LIN {X 0,Y 542.795,Z 373.704,A -85,B 0,C 180,E1 23564.562,E2 23564.562} C_VEL
LIN {X 0,Y 545.816,Z 376.25,A -85,B 0,C 180,E1 23563.586,E2 23563.586} C_VEL
LIN {X 0,Y 548.815,Z 380.332,A -85,B 0,C 180,E1 23562.615,E2 23562.615} C_VEL
LIN {X 0,Y 551.245,Z 382.532,A -85,B 0,C 180,E1 23561.903,E2 23561.903} C_VEL
LIN {X 0,Y 554.687,Z 386.919,A -85,B 0,C 180,E1 23560.902,E2 23560.902} C_VEL
LIN {X 0,Y 556.558,Z 388.828,A -85,B 0,C 180,E1 23560.396,E2 23560.396} C_VEL
LIN {X 0,Y 560.439,Z 393.498,A -85,B 0,C 180,E1 23559.368,E2 23559.368} C_VEL
LIN {X 0,Y 566.505,Z 400.97,A -85,B 0,C 180,E1 23557.862,E2 23557.862} C_VEL
LIN {X 0,Y 571.785,Z 407.602,A -85,B 0,C 180,E1 23556.639,E2 23556.639} C_VEL
LIN {X 0,Y 577.51,Z 414.886,A -85,B 0,C 180,E1 23555.392,E2 23555.392} C_VEL
LIN {X 0,Y 587.049,Z 428.51,A -85,B 0,C 180,E1 23553.442,E2 23553.442} C_VEL
LIN {X 0,Y 595.115,Z 441.003,A -85,B 0,C 180,E1 23551.909,E2 23551.909} C_VEL
LIN {X 0,Y 595.96,Z 442.638,A -85,B 0,C 180,E1 23551.748,E2 23551.748} C_VEL
LIN {X 0,Y 586.943,Z 655.568,A -85,B 0,C 180,E1 23548.557,E2 23548.557} C_VEL
LIN {X 0,Y 580.387,Z 818.11,A -85,B 0,C 180,E1 23546.144,E2 23546.144} C_VEL
LIN {X 0,Y 578.548,Z 843.182,A -85,B 0,C 180,E1 23545.671,E2 23545.671} C_VEL
LIN {X 0,Y 575.71,Z 870.919,A -85,B 0,C 180,E1 23544.956,E2 23544.956} C_VEL
LIN {X 0,Y 573.073,Z 892.207,A -85,B 0,C 180,E1 23544.266,E2 23544.266} C_VEL
LIN {X 0,Y 570.199,Z 912.697,A -85,B 0,C 180,E1 23543.475,E2 23543.475} C_VEL
LIN {X 0,Y 567.095,Z 932.487,A -85,B 0,C 180,E1 23542.588,E2 23542.588} C_VEL
LIN {X 0,Y 564.019,Z 950.451,A -85,B 0,C 180,E1 23541.669,E2 23541.669} C_VEL
LIN {X 0,Y 562.069,Z 957.506,A -85,B 0,C 180,E1 23541.362,E2 23541.362} C_VEL
LIN {X 0,Y 554.369,Z 974.984,A -85,B 0,C 180,E1 23540.75,E2 23540.75} C_VEL
LIN {X 0,Y 552.285,Z 981.526,A -85,B 0,C 180,E1 23540.385,E2 23540.385} C_VEL
LIN {X 0,Y 548.266,Z 1000.587,A -85,B 0,C 180,E1 23539.025,E2 23539.025} C_VEL
LIN {X 0,Y 544.207,Z 1019.207,A -85,B 0,C 180,E1 23537.533,E2 23537.533} C_VEL
LIN {X 0,Y 539.48,Z 1040.477,A -85,B 0,C 180,E1 23535.6,E2 23535.6} C_VEL
LIN {X 0,Y 534.654,Z 1061.325,A -85,B 0,C 180,E1 23533.414,E2 23533.414} C_VEL
LIN {X 0,Y 530.182,Z 1080.685,A -85,B 0,C 180,E1 23531.091,E2 23531.091} C_VEL
LIN {X 0,Y 526.071,Z 1099.032,A -85,B 0,C 180,E1 23528.565,E2 23528.565} C_VEL
LIN {X 0,Y 522.347,Z 1116.161,A -85,B 0,C 180,E1 23525.855,E2 23525.855} C_VEL
LIN {X 0,Y 519.741,Z 1129.22,A -85,B 0,C 180,E1 23523.512,E2 23523.512} C_VEL
LIN {X 0,Y 517.517,Z 1141.407,A -85,B 0,C 180,E1 23521.054,E2 23521.054} C_VEL
LIN {X 0,Y 515.395,Z 1154.516,A -85,B 0,C 180,E1 23518,E2 23518} C_VEL
LIN {X 0,Y 514.05,Z 1164.255,A -85,B 0,C 180,E1 23515.335,E2 23515.335} C_VEL
LIN {X 0,Y 513.094,Z 1172.905,A -85,B 0,C 180,E1 23512.575,E2 23512.575} C_VEL
LIN {X 0,Y 512.416,Z 1180.779,A -85,B 0,C 180,E1 23509.491,E2 23509.491} C_VEL
LIN {X 0,Y 512.131,Z 1185.993,A -85,B 0,C 180,E1 23506.912,E2 23506.912} C_VEL
LIN {X 0,Y 511.987,Z 1189.961,A -85,B 0,C 180,E1 23504.379,E2 23504.379} C_VEL
LIN {X 0,Y 511.919,Z 1193.03,A -85,B 0,C 180,E1 23501.606,E2 23501.606} C_VEL
LIN {X 0,Y 511.91,Z 1194.672,A -85,B 0,C 180,E1 23498.65,E2 23498.65} C_VEL
LIN {X 0,Y 511.913,Z 1194.851,A -85,B 0,C 180,E1 23496.167,E2 23496.167} C_VEL
LIN {X 0,Y 511.909,Z 1193.96,A -85,B 0,C 180,E1 23493.696,E2 23493.696} C_VEL
LIN {X 0,Y 511.935,Z 1191.975,A -85,B 0,C 180,E1 23491.231,E2 23491.231} C_VEL
LIN {X 0,Y 512.028,Z 1188.452,A -85,B 0,C 180,E1 23488.433,E2 23488.433} C_VEL
LIN {X 0,Y 512.288,Z 1182.928,A -85,B 0,C 180,E1 23485.41,E2 23485.41} C_VEL
LIN {X 0,Y 512.716,Z 1176.911,A -85,B 0,C 180,E1 23482.83,E2 23482.83} C_VEL
LIN {X 0,Y 513.428,Z 1169.662,A -85,B 0,C 180,E1 23480.246,E2 23480.246} C_VEL
LIN {X 0,Y 514.741,Z 1159.044,A -85,B 0,C 180,E1 23477.092,E2 23477.092} C_VEL
LIN {X 0,Y 516.276,Z 1148.691,A -85,B 0,C 180,E1 23474.499,E2 23474.499} C_VEL
LIN {X 0,Y 518.205,Z 1137.424,A -85,B 0,C 180,E1 23472.018,E2 23472.018} C_VEL
LIN {X 0,Y 521.153,Z 1122.163,A -85,B 0,C 180,E1 23469.093,E2 23469.093} C_VEL
LIN {X 0,Y 524.187,Z 1107.393,A -85,B 0,C 180,E1 23466.625,E2 23466.625} C_VEL
LIN {X 0,Y 527.705,Z 1091.651,A -85,B 0,C 180,E1 23464.285,E2 23464.285} C_VEL
LIN {X 0,Y 532.183,Z 1072.006,A -85,B 0,C 180,E1 23461.741,E2 23461.741} C_VEL
LIN {X 0,Y 536.871,Z 1051.612,A -85,B 0,C 180,E1 23459.441,E2 23459.441} C_VEL
LIN {X 0,Y 541.664,Z 1030.618,A -85,B 0,C 180,E1 23457.384,E2 23457.384} C_VEL
LIN {X 0,Y 546.846,Z 1007.416,A -85,B 0,C 180,E1 23455.409,E2 23455.409} C_VEL
LIN {X 0,Y 551.213,Z 986.563,A -85,B 0,C 180,E1 23453.877,E2 23453.877} C_VEL
LIN {X 0,Y 554.892,Z 968.037,A -85,B 0,C 180,E1 23452.675,E2 23452.675} C_VEL
LIN {X 0,Y 558.395,Z 949.059,A -85,B 0,C 180,E1 23451.586,E2 23451.586} C_VEL
LIN {X 0,Y 561.883,Z 928.574,A -85,B 0,C 180,E1 23450.56,E2 23450.56} C_VEL
LIN {X 0,Y 565.837,Z 903.019,A -85,B 0,C 180,E1 23449.471,E2 23449.471} C_VEL
LIN {X 0,Y 569.101,Z 877.277,A -85,B 0,C 180,E1 23448.59,E2 23448.59} C_VEL
LIN {X 0,Y 571.431,Z 855.733,A -85,B 0,C 180,E1 23447.989,E2 23447.989} C_VEL
LIN {X 0,Y 573.333,Z 834.31,A -85,B 0,C 180,E1 23447.511,E2 23447.511} C_VEL
LIN {X 0,Y 574.879,Z 810.042,A -85,B 0,C 180,E1 23447.093,E2 23447.093} C_VEL
LIN {X 0,Y 582.975,Z 592.298,A -85,B 0,C 180,E1 23443.915,E2 23443.915} C_VEL
LIN {X 0,Y 588.599,Z 446.247,A -85,B 0,C 180,E1 23441.753,E2 23441.753} C_VEL
LIN {X 0,Y 572.418,Z 422.974,A -85,B 0,C 180,E1 23439.029,E2 23439.029} C_VEL
LIN {X 0,Y 564.92,Z 412.761,A -85,B 0,C 180,E1 23437.668,E2 23437.668} C_VEL
LIN {X 0,Y 556.568,Z 402.056,A -85,B 0,C 180,E1 23436.067,E2 23436.067} C_VEL
LIN {X 0,Y 548.839,Z 392.277,A -85,B 0,C 180,E1 23434.481,E2 23434.481} C_VEL
LIN {X 0,Y 543.88,Z 386.332,A -85,B 0,C 180,E1 23433.409,E2 23433.409} C_VEL
LIN {X 0,Y 539.41,Z 380.867,A -85,B 0,C 180,E1 23432.392,E2 23432.392} C_VEL
LIN {X 0,Y 535.79,Z 376.492,A -85,B 0,C 180,E1 23431.534,E2 23431.534} C_VEL
LIN {X 0,Y 534.25,Z 374.853,A -85,B 0,C 180,E1 23431.164,E2 23431.164} C_VEL
LIN {X 0,Y 530.972,Z 370.926,A -85,B 0,C 180,E1 23430.342,E2 23430.342} C_VEL
LIN {X 0,Y 529.918,Z 369.476,A -85,B 0,C 180,E1 23430.064,E2 23430.064} C_VEL
LIN {X 0,Y 526.592,Z 366.343,A -85,B 0,C 180,E1 23429.209,E2 23429.209} C_VEL
LIN {X 0,Y 524.818,Z 363.288,A -85,B 0,C 180,E1 23428.693,E2 23428.693} C_VEL
LIN {X 0,Y 521.507,Z 360.788,A -85,B 0,C 180,E1 23427.8,E2 23427.8} C_VEL
LIN {X 0,Y 519.538,Z 357.406,A -85,B 0,C 180,E1 23427.184,E2 23427.184} C_VEL
LIN {X 0,Y 519.072,Z 356.737,A -85,B 0,C 180,E1 23427.04,E2 23427.04} C_VEL
LIN {X 0,Y 515.845,Z 354.704,A -85,B 0,C 180,E1 23426.104,E2 23426.104} C_VEL
LIN {X 0,Y 514.186,Z 351.972,A -85,B 0,C 180,E1 23425.542,E2 23425.542} C_VEL
LIN {X 0,Y 513.777,Z 350.215,A -85,B 0,C 180,E1 23425.351,E2 23425.351} C_VEL
LIN {X 0,Y 513.713,Z 350.161,A -85,B 0,C 180,E1 23422.065,E2 23422.065} C_VEL
LIN {X 0,Y 513.745,Z 350.236,A -85,B 0,C 180,E1 23418.614,E2 23418.614} C_VEL
LIN {X 0,Y 513.754,Z 350.233,A -85,B 0,C 180,E1 23415.349,E2 23415.349} C_VEL
LIN {X 0,Y 513.723,Z 350.235,A -85,B 0,C 180,E1 23412.021,E2 23412.021} C_VEL
LIN {X 0,Y 513.776,Z 350.224,A -85,B 0,C 180,E1 23408.619,E2 23408.619} C_VEL
LIN {X 0,Y 513.734,Z 350.224,A -85,B 0,C 180,E1 23405.361,E2 23405.361} C_VEL
LIN {X 0,Y 513.728,Z 350.224,A -85,B 0,C 180,E1 23401.896,E2 23401.896} C_VEL
LIN {X 0,Y 513.784,Z 350.213,A -85,B 0,C 180,E1 23398.662,E2 23398.662} C_VEL
LIN {X 0,Y 513.727,Z 350.218,A -85,B 0,C 180,E1 23395.311,E2 23395.311} C_VEL
LIN {X 0,Y 513.743,Z 350.219,A -85,B 0,C 180,E1 23391.832,E2 23391.832} C_VEL
LIN {X 0,Y 513.764,Z 350.175,A -85,B 0,C 180,E1 23388.55,E2 23388.55} C_VEL
LIN {X 0,Y 513.725,Z 350.191,A -85,B 0,C 180,E1 23385.228,E2 23385.228} C_VEL
LIN {X 0,Y 513.781,Z 350.168,A -85,B 0,C 180,E1 23381.975,E2 23381.975} C_VEL
LIN {X 0,Y 513.776,Z 350.304,A -85,B 0,C 180,E1 23381.74,E2 23381.74} C_VEL
LIN {X 0,Y 514.652,Z 353.02,A -85,B 0,C 180,E1 23381.391,E2 23381.391} C_VEL
LIN {X 0,Y 516.89,Z 355.586,A -85,B 0,C 180,E1 23380.683,E2 23380.683} C_VEL
LIN {X 0,Y 519.415,Z 357.122,A -85,B 0,C 180,E1 23379.961,E2 23379.961} C_VEL
LIN {X 0,Y 521.3,Z 360.559,A -85,B 0,C 180,E1 23379.363,E2 23379.363} C_VEL
LIN {X 0,Y 524.371,Z 363.099,A -85,B 0,C 180,E1 23378.524,E2 23378.524} C_VEL
LIN {X 0,Y 525.111,Z 363.904,A -85,B 0,C 180,E1 23378.321,E2 23378.321} C_VEL
LIN {X 0,Y 527.649,Z 367.603,A -85,B 0,C 180,E1 23377.611,E2 23377.611} C_VEL
LIN {X 0,Y 530.517,Z 370.117,A -85,B 0,C 180,E1 23376.887,E2 23376.887} C_VEL
LIN {X 0,Y 533.502,Z 374.128,A -85,B 0,C 180,E1 23376.12,E2 23376.12} C_VEL
LIN {X 0,Y 535.754,Z 376.327,A -85,B 0,C 180,E1 23375.582,E2 23375.582} C_VEL
LIN {X 0,Y 545.223,Z 388.341,A -85,B 0,C 180,E1 23373.389,E2 23373.389} C_VEL
LIN {X 0,Y 553.809,Z 399.693,A -85,B 0,C 180,E1 23371.563,E2 23371.563} C_VEL
LIN {X 0,Y 562.926,Z 412.152,A -85,B 0,C 180,E1 23369.764,E2 23369.764} C_VEL
LIN {X 0,Y 575.646,Z 430.28,A -85,B 0,C 180,E1 23367.45,E2 23367.45} C_VEL
LIN {X 0,Y 588.662,Z 449.546,A -85,B 0,C 180,E1 23365.278,E2 23365.278} C_VEL
LIN {X 0,Y 580.389,Z 665.721,A -85,B 0,C 180,E1 23362.096,E2 23362.096} C_VEL
LIN {X 0,Y 574.374,Z 825.899,A -85,B 0,C 180,E1 23359.751,E2 23359.751} C_VEL
LIN {X 0,Y 572.583,Z 850.667,A -85,B 0,C 180,E1 23359.295,E2 23359.295} C_VEL
LIN {X 0,Y 569.722,Z 879.093,A -85,B 0,C 180,E1 23358.578,E2 23358.578} C_VEL
LIN {X 0,Y 567.068,Z 900.639,A -85,B 0,C 180,E1 23357.891,E2 23357.891} C_VEL
LIN {X 0,Y 564.208,Z 921.045,A -85,B 0,C 180,E1 23357.115,E2 23357.115} C_VEL
LIN {X 0,Y 560.986,Z 941.539,A -85,B 0,C 180,E1 23356.206,E2 23356.206} C_VEL
LIN {X 0,Y 556.988,Z 964.689,A -85,B 0,C 180,E1 23355.013,E2 23355.013} C_VEL
LIN {X 0,Y 552.164,Z 989.777,A -85,B 0,C 180,E1 23353.48,E2 23353.48} C_VEL
LIN {X 0,Y 548.264,Z 1008.64,A -85,B 0,C 180,E1 23352.153,E2 23352.153} C_VEL
LIN {X 0,Y 544.316,Z 1026.981,A -85,B 0,C 180,E1 23350.7,E2 23350.7} C_VEL
LIN {X 0,Y 540.243,Z 1045.39,A -85,B 0,C 180,E1 23349.063,E2 23349.063} C_VEL
LIN {X 0,Y 535.325,Z 1067.373,A -85,B 0,C 180,E1 23346.838,E2 23346.838} C_VEL
LIN {X 0,Y 531.26,Z 1085.19,A -85,B 0,C 180,E1 23344.768,E2 23344.768} C_VEL
LIN {X 0,Y 528.053,Z 1099.503,A -85,B 0,C 180,E1 23342.917,E2 23342.917} C_VEL
LIN {X 0,Y 525.031,Z 1113.29,A -85,B 0,C 180,E1 23340.943,E2 23340.943} C_VEL
LIN {X 0,Y 522.121,Z 1127.167,A -85,B 0,C 180,E1 23338.729,E2 23338.729} C_VEL
LIN {X 0,Y 519.005,Z 1143.116,A -85,B 0,C 180,E1 23335.81,E2 23335.81} C_VEL
LIN {X 0,Y 516.929,Z 1154.738,A -85,B 0,C 180,E1 23333.36,E2 23333.36} C_VEL
LIN {X 0,Y 515.373,Z 1164.516,A -85,B 0,C 180,E1 23331.033,E2 23331.033} C_VEL
LIN {X 0,Y 514.198,Z 1173.103,A -85,B 0,C 180,E1 23328.714,E2 23328.714} C_VEL
LIN {X 0,Y 513.172,Z 1181.977,A -85,B 0,C 180,E1 23325.945,E2 23325.945} C_VEL
LIN {X 0,Y 512.473,Z 1190.05,A -85,B 0,C 180,E1 23322.851,E2 23322.851} C_VEL
LIN {X 0,Y 512.147,Z 1195.486,A -85,B 0,C 180,E1 23320.233,E2 23320.233} C_VEL
LIN {X 0,Y 511.999,Z 1199.358,A -85,B 0,C 180,E1 23317.857,E2 23317.857} C_VEL
LIN {X 0,Y 511.932,Z 1202.314,A -85,B 0,C 180,E1 23315.379,E2 23315.379} C_VEL
LIN {X 0,Y 511.912,Z 1204.305,A -85,B 0,C 180,E1 23312.687,E2 23312.687} C_VEL
LIN {X 0,Y 511.897,Z 1204.939,A -85,B 0,C 180,E1 23309.664,E2 23309.664} C_VEL
LIN {X 0,Y 511.916,Z 1204.1,A -85,B 0,C 180,E1 23306.977,E2 23306.977} C_VEL
LIN {X 0,Y 511.933,Z 1202.199,A -85,B 0,C 180,E1 23304.508,E2 23304.508} C_VEL
LIN {X 0,Y 512.006,Z 1199.197,A -85,B 0,C 180,E1 23302.03,E2 23302.03} C_VEL
LIN {X 0,Y 512.169,Z 1195.073,A -85,B 0,C 180,E1 23299.54,E2 23299.54} C_VEL
LIN {X 0,Y 512.613,Z 1188.472,A -85,B 0,C 180,E1 23296.464,E2 23296.464} C_VEL
LIN {X 0,Y 513.312,Z 1180.562,A -85,B 0,C 180,E1 23293.594,E2 23293.594} C_VEL
LIN {X 0,Y 514.249,Z 1172.698,A -85,B 0,C 180,E1 23291.17,E2 23291.17} C_VEL
LIN {X 0,Y 515.439,Z 1164.061,A -85,B 0,C 180,E1 23288.85,E2 23288.85} C_VEL
LIN {X 0,Y 517.113,Z 1153.715,A -85,B 0,C 180,E1 23286.407,E2 23286.407} C_VEL
LIN {X 0,Y 519.812,Z 1138.894,A -85,B 0,C 180,E1 23283.373,E2 23283.373} C_VEL
LIN {X 0,Y 522.451,Z 1125.546,A -85,B 0,C 180,E1 23281.001,E2 23281.001} C_VEL
LIN {X 0,Y 525.203,Z 1112.507,A -85,B 0,C 180,E1 23278.941,E2 23278.941} C_VEL
LIN {X 0,Y 528.242,Z 1098.637,A -85,B 0,C 180,E1 23276.967,E2 23276.967} C_VEL
LIN {X 0,Y 532.231,Z 1080.973,A -85,B 0,C 180,E1 23274.713,E2 23274.713} C_VEL
LIN {X 0,Y 536.861,Z 1060.276,A -85,B 0,C 180,E1 23272.415,E2 23272.415} C_VEL
LIN {X 0,Y 540.77,Z 1042.882,A -85,B 0,C 180,E1 23270.709,E2 23270.709} C_VEL
LIN {X 0,Y 544.733,Z 1024.943,A -85,B 0,C 180,E1 23269.135,E2 23269.135} C_VEL
LIN {X 0,Y 549.73,Z 1001.929,A -85,B 0,C 180,E1 23267.351,E2 23267.351} C_VEL
LIN {X 0,Y 554.397,Z 978.674,A -85,B 0,C 180,E1 23265.809,E2 23265.809} C_VEL
LIN {X 0,Y 558.111,Z 959.029,A -85,B 0,C 180,E1 23264.665,E2 23264.665} C_VEL
LIN {X 0,Y 561.651,Z 938.954,A -85,B 0,C 180,E1 23263.643,E2 23263.643} C_VEL
LIN {X 0,Y 565.072,Z 917.752,A -85,B 0,C 180,E1 23262.71,E2 23262.71} C_VEL
LIN {X 0,Y 568.897,Z 890.935,A -85,B 0,C 180,E1 23261.725,E2 23261.725} C_VEL
LIN {X 0,Y 571.809,Z 865.86,A -85,B 0,C 180,E1 23261.001,E2 23261.001} C_VEL
LIN {X 0,Y 573.885,Z 844.227,A -85,B 0,C 180,E1 23260.507,E2 23260.507} C_VEL
LIN {X 0,Y 575.468,Z 821.977,A -85,B 0,C 180,E1 23260.11,E2 23260.11} C_VEL
LIN {X 0,Y 584.635,Z 602.928,A -85,B 0,C 180,E1 23256.842,E2 23256.842} C_VEL
LIN {X 0,Y 591.403,Z 449.585,A -85,B 0,C 180,E1 23254.516,E2 23254.516} C_VEL
LIN {X 0,Y 582.117,Z 434.895,A -85,B 0,C 180,E1 23252.692,E2 23252.692} C_VEL
LIN {X 0,Y 571.453,Z 419.408,A -85,B 0,C 180,E1 23250.405,E2 23250.405} C_VEL
LIN {X 0,Y 562.947,Z 408.071,A -85,B 0,C 180,E1 23248.397,E2 23248.397} C_VEL
LIN {X 0,Y 559.293,Z 403.321,A -85,B 0,C 180,E1 23247.468,E2 23247.468} C_VEL
LIN {X 0,Y 554.987,Z 397.689,A -85,B 0,C 180,E1 23246.309,E2 23246.309} C_VEL
LIN {X 0,Y 550.544,Z 392.044,A -85,B 0,C 180,E1 23245.035,E2 23245.035} C_VEL
LIN {X 0,Y 547.278,Z 388.136,A -85,B 0,C 180,E1 23244.043,E2 23244.043} C_VEL
LIN {X 0,Y 543.121,Z 382.967,A -85,B 0,C 180,E1 23242.687,E2 23242.687} C_VEL
LIN {X 0,Y 539.863,Z 379.736,A -85,B 0,C 180,E1 23241.571,E2 23241.571} C_VEL
LIN {X 0,Y 538.134,Z 376.988,A -85,B 0,C 180,E1 23240.901,E2 23240.901} C_VEL
LIN {X 0,Y 534.85,Z 374.402,A -85,B 0,C 180,E1 23239.664,E2 23239.664} C_VEL
LIN {X 0,Y 532.518,Z 370.548,A -85,B 0,C 180,E1 23238.615,E2 23238.615} C_VEL
LIN {X 0,Y 528.86,Z 367.985,A -85,B 0,C 180,E1 23236.984,E2 23236.984} C_VEL
LIN {X 0,Y 526.971,Z 364.842,A -85,B 0,C 180,E1 23235.941,E2 23235.941} C_VEL
LIN {X 0,Y 526.483,Z 363.856,A -85,B 0,C 180,E1 23235.646,E2 23235.646} C_VEL
LIN {X 0,Y 523.26,Z 362.124,A -85,B 0,C 180,E1 23233.819,E2 23233.819} C_VEL
LIN {X 0,Y 521.056,Z 359.128,A -85,B 0,C 180,E1 23232.186,E2 23232.186} C_VEL
LIN {X 0,Y 520.346,Z 357.063,A -85,B 0,C 180,E1 23231.485,E2 23231.485} C_VEL
LIN {X 0,Y 515.465,Z 354.269,A -85,B 0,C 180,E1 23224.339,E2 23224.339} C_VEL
LIN {X 0,Y 515.79,Z 354.54,A -85,B 0,C 180,E1 23221.111,E2 23221.111} C_VEL
LIN {X 0,Y 520.495,Z 357.25,A -85,B 0,C 180,E1 23215.179,E2 23215.179} C_VEL
LIN {X 0,Y 521.575,Z 360.156,A -85,B 0,C 180,E1 23214.168,E2 23214.168} C_VEL
LIN {X 0,Y 524.682,Z 363.149,A -85,B 0,C 180,E1 23212.113,E2 23212.113} C_VEL
LIN {X 0,Y 526.72,Z 364.108,A -85,B 0,C 180,E1 23211.017,E2 23211.017} C_VEL
LIN {X 0,Y 528.427,Z 367.464,A -85,B 0,C 180,E1 23210.03,E2 23210.03} C_VEL
LIN {X 0,Y 531.73,Z 370.227,A -85,B 0,C 180,E1 23208.502,E2 23208.502} C_VEL
LIN {X 0,Y 532.836,Z 371.044,A -85,B 0,C 180,E1 23208.032,E2 23208.032} C_VEL
LIN {X 0,Y 535.199,Z 374.766,A -85,B 0,C 180,E1 23206.99,E2 23206.99} C_VEL
LIN {X 0,Y 538.495,Z 377.417,A -85,B 0,C 180,E1 23205.757,E2 23205.757} C_VEL
LIN {X 0,Y 541.222,Z 381.379,A -85,B 0,C 180,E1 23204.736,E2 23204.736} C_VEL
LIN {X 0,Y 544.046,Z 383.878,A -85,B 0,C 180,E1 23203.805,E2 23203.805} C_VEL
LIN {X 0,Y 547.184,Z 388.01,A -85,B 0,C 180,E1 23202.781,E2 23202.781} C_VEL
LIN {X 0,Y 549.412,Z 390.163,A -85,B 0,C 180,E1 23202.115,E2 23202.115} C_VEL
LIN {X 0,Y 553.006,Z 394.601,A -85,B 0,C 180,E1 23201.061,E2 23201.061} C_VEL
LIN {X 0,Y 554.752,Z 396.587,A -85,B 0,C 180,E1 23200.577,E2 23200.577} C_VEL
LIN {X 0,Y 559.98,Z 402.962,A -85,B 0,C 180,E1 23199.186,E2 23199.186} C_VEL
LIN {X 0,Y 564.427,Z 408.477,A -85,B 0,C 180,E1 23198.078,E2 23198.078} C_VEL
LIN {X 0,Y 570.065,Z 415.607,A -85,B 0,C 180,E1 23196.756,E2 23196.756} C_VEL
LIN {X 0,Y 576.376,Z 423.908,A -85,B 0,C 180,E1 23195.368,E2 23195.368} C_VEL
LIN {X 0,Y 586.787,Z 439.139,A -85,B 0,C 180,E1 23193.238,E2 23193.238} C_VEL
LIN {X 0,Y 591.421,Z 446.898,A -85,B 0,C 180,E1 23192.337,E2 23192.337} C_VEL
LIN {X 0,Y 582.041,Z 659.407,A -85,B 0,C 180,E1 23189.136,E2 23189.136} C_VEL
LIN {X 0,Y 575.336,Z 818.273,A -85,B 0,C 180,E1 23186.762,E2 23186.762} C_VEL
LIN {X 0,Y 573.4,Z 843.673,A -85,B 0,C 180,E1 23186.28,E2 23186.28} C_VEL
LIN {X 0,Y 570.475,Z 871.11,A -85,B 0,C 180,E1 23185.568,E2 23185.568} C_VEL
LIN {X 0,Y 567.662,Z 892.917,A -85,B 0,C 180,E1 23184.856,E2 23184.856} C_VEL
LIN {X 0,Y 564.683,Z 913.265,A -85,B 0,C 180,E1 23184.064,E2 23184.064} C_VEL
LIN {X 0,Y 561.457,Z 932.937,A -85,B 0,C 180,E1 23183.176,E2 23183.176} C_VEL
LIN {X 0,Y 557.311,Z 956.133,A -85,B 0,C 180,E1 23181.961,E2 23181.961} C_VEL
LIN {X 0,Y 552.389,Z 981.023,A -85,B 0,C 180,E1 23180.419,E2 23180.419} C_VEL
LIN {X 0,Y 552.285,Z 981.526,A -85,B 0,C 180,E1 23180.385,E2 23180.385} C_VEL
LIN {X 0,Y 550.201,Z 988.111,A -85,B 0,C 180,E1 23180.008,E2 23180.008} C_VEL
LIN {X 0,Y 541.717,Z 1005.826,A -85,B 0,C 180,E1 23179.172,E2 23179.172} C_VEL
LIN {X 0,Y 539.884,Z 1011.139,A -85,B 0,C 180,E1 23178.797,E2 23178.797} C_VEL
LIN {X 0,Y 535.021,Z 1031.788,A -85,B 0,C 180,E1 23176.988,E2 23176.988} C_VEL
LIN {X 0,Y 530.799,Z 1049.476,A -85,B 0,C 180,E1 23175.247,E2 23175.247} C_VEL
LIN {X 0,Y 526.163,Z 1068.801,A -85,B 0,C 180,E1 23173.098,E2 23173.098} C_VEL
LIN {X 0,Y 521.401,Z 1088.672,A -85,B 0,C 180,E1 23170.547,E2 23170.547} C_VEL
LIN {X 0,Y 517.416,Z 1105.609,A -85,B 0,C 180,E1 23168.056,E2 23168.056} C_VEL
LIN {X 0,Y 514.103,Z 1120.509,A -85,B 0,C 180,E1 23165.557,E2 23165.557} C_VEL
LIN {X 0,Y 510.897,Z 1136.144,A -85,B 0,C 180,E1 23162.561,E2 23162.561} C_VEL
LIN {X 0,Y 508.724,Z 1147.939,A -85,B 0,C 180,E1 23159.948,E2 23159.948} C_VEL
LIN {X 0,Y 507.12,Z 1157.792,A -85,B 0,C 180,E1 23157.468,E2 23157.468} C_VEL
LIN {X 0,Y 505.709,Z 1168.269,A -85,B 0,C 180,E1 23154.407,E2 23154.407} C_VEL
LIN {X 0,Y 504.861,Z 1176.127,A -85,B 0,C 180,E1 23151.615,E2 23151.615} C_VEL
LIN {X 0,Y 504.377,Z 1182.056,A -85,B 0,C 180,E1 23149.092,E2 23149.092} C_VEL
LIN {X 0,Y 504.1,Z 1187.026,A -85,B 0,C 180,E1 23146.477,E2 23146.477} C_VEL
LIN {X 0,Y 503.954,Z 1191.34,A -85,B 0,C 180,E1 23143.423,E2 23143.423} C_VEL
LIN {X 0,Y 503.916,Z 1193.744,A -85,B 0,C 180,E1 23140.634,E2 23140.634} C_VEL
LIN {X 0,Y 503.91,Z 1194.762,A -85,B 0,C 180,E1 23138.214,E2 23138.214} C_VEL
LIN {X 0,Y 503.913,Z 1194.806,A -85,B 0,C 180,E1 23135.922,E2 23135.922} C_VEL
LIN {X 0,Y 503.911,Z 1193.89,A -85,B 0,C 180,E1 23133.527,E2 23133.527} C_VEL
LIN {X 0,Y 503.944,Z 1191.749,A -85,B 0,C 180,E1 23130.909,E2 23130.909} C_VEL
LIN {X 0,Y 504.071,Z 1187.737,A -85,B 0,C 180,E1 23127.84,E2 23127.84} C_VEL
LIN {X 0,Y 504.35,Z 1182.436,A -85,B 0,C 180,E1 23124.996,E2 23124.996} C_VEL
LIN {X 0,Y 504.798,Z 1176.618,A -85,B 0,C 180,E1 23122.488,E2 23122.488} C_VEL
LIN {X 0,Y 505.573,Z 1169.325,A -85,B 0,C 180,E1 23119.862,E2 23119.862} C_VEL
LIN {X 0,Y 507.014,Z 1158.61,A -85,B 0,C 180,E1 23116.66,E2 23116.66} C_VEL
LIN {X 0,Y 508.578,Z 1148.692,A -85,B 0,C 180,E1 23114.141,E2 23114.141} C_VEL
LIN {X 0,Y 510.514,Z 1137.964,A -85,B 0,C 180,E1 23111.738,E2 23111.738} C_VEL
LIN {X 0,Y 513.53,Z 1123.335,A -85,B 0,C 180,E1 23108.854,E2 23108.854} C_VEL
LIN {X 0,Y 516.964,Z 1107.5,A -85,B 0,C 180,E1 23106.157,E2 23106.157} C_VEL
LIN {X 0,Y 520.857,Z 1090.921,A -85,B 0,C 180,E1 23103.677,E2 23103.677} C_VEL
LIN {X 0,Y 525.36,Z 1072.114,A -85,B 0,C 180,E1 23101.216,E2 23101.216} C_VEL
LIN {X 0,Y 530.323,Z 1051.443,A -85,B 0,C 180,E1 23098.87,E2 23098.87} C_VEL
LIN {X 0,Y 534.853,Z 1032.405,A -85,B 0,C 180,E1 23096.98,E2 23096.98} C_VEL
LIN {X 0,Y 539.606,Z 1012.096,A -85,B 0,C 180,E1 23095.201,E2 23095.201} C_VEL
LIN {X 0,Y 544.887,Z 988.086,A -85,B 0,C 180,E1 23093.39,E2 23093.39} C_VEL
LIN {X 0,Y 548.852,Z 968.788,A -85,B 0,C 180,E1 23092.127,E2 23092.127} C_VEL
LIN {X 0,Y 552.473,Z 949.827,A -85,B 0,C 180,E1 23091.031,E2 23091.031} C_VEL
LIN {X 0,Y 556.082,Z 929.312,A -85,B 0,C 180,E1 23089.996,E2 23089.996} C_VEL
LIN {X 0,Y 559.848,Z 905.752,A -85,B 0,C 180,E1 23088.979,E2 23088.979} C_VEL
LIN {X 0,Y 563.497,Z 878.515,A -85,B 0,C 180,E1 23088.026,E2 23088.026} C_VEL
LIN {X 0,Y 565.972,Z 856.417,A -85,B 0,C 180,E1 23087.403,E2 23087.403} C_VEL
LIN {X 0,Y 567.944,Z 834.944,A -85,B 0,C 180,E1 23086.921,E2 23086.921} C_VEL
LIN {X 0,Y 569.497,Z 811.607,A -85,B 0,C 180,E1 23086.514,E2 23086.514} C_VEL
LIN {X 0,Y 577.796,Z 596.882,A -85,B 0,C 180,E1 23083.361,E2 23083.361} C_VEL
LIN {X 0,Y 583.632,Z 450.363,A -85,B 0,C 180,E1 23081.179,E2 23081.179} C_VEL
LIN {X 0,Y 565.947,Z 424.806,A -85,B 0,C 180,E1 23078.101,E2 23078.101} C_VEL
LIN {X 0,Y 554.743,Z 410.081,A -85,B 0,C 180,E1 23075.955,E2 23075.955} C_VEL
LIN {X 0,Y 545.35,Z 398.347,A -85,B 0,C 180,E1 23074.002,E2 23074.002} C_VEL
LIN {X 0,Y 541.332,Z 393.389,A -85,B 0,C 180,E1 23073.112,E2 23073.112} C_VEL
LIN {X 0,Y 536.734,Z 387.788,A -85,B 0,C 180,E1 23072.049,E2 23072.049} C_VEL
LIN {X 0,Y 532.32,Z 382.419,A -85,B 0,C 180,E1 23070.976,E2 23070.976} C_VEL
LIN {X 0,Y 528.666,Z 378.133,A -85,B 0,C 180,E1 23070.049,E2 23070.049} C_VEL
LIN {X 0,Y 527.414,Z 376.629,A -85,B 0,C 180,E1 23069.72,E2 23069.72} C_VEL
LIN {X 0,Y 523.977,Z 372.997,A -85,B 0,C 180,E1 23068.806,E2 23068.806} C_VEL
LIN {X 0,Y 522.372,Z 370.594,A -85,B 0,C 180,E1 23068.34,E2 23068.34} C_VEL
LIN {X 0,Y 519.059,Z 367.632,A -85,B 0,C 180,E1 23067.413,E2 23067.413} C_VEL
LIN {X 0,Y 517.07,Z 364.341,A -85,B 0,C 180,E1 23066.78,E2 23066.78} C_VEL
LIN {X 0,Y 513.902,Z 362.09,A -85,B 0,C 180,E1 23065.838,E2 23065.838} C_VEL
LIN {X 0,Y 511.885,Z 358.784,A -85,B 0,C 180,E1 23065.142,E2 23065.142} C_VEL
LIN {X 0,Y 511.444,Z 357.891,A -85,B 0,C 180,E1 23064.979,E2 23064.979} C_VEL
LIN {X 0,Y 508.316,Z 356.108,A -85,B 0,C 180,E1 23063.966,E2 23063.966} C_VEL
LIN {X 0,Y 506.442,Z 353.358,A -85,B 0,C 180,E1 23063.258,E2 23063.258} C_VEL
LIN {X 0,Y 505.815,Z 351.156,A -85,B 0,C 180,E1 23062.919,E2 23062.919} C_VEL
LIN {X 0,Y 505.796,Z 351.182,A -85,B 0,C 180,E1 23059.638,E2 23059.638} C_VEL
LIN {X 0,Y 505.783,Z 351.211,A -85,B 0,C 180,E1 23056.185,E2 23056.185} C_VEL
LIN {X 0,Y 505.846,Z 351.202,A -85,B 0,C 180,E1 23052.907,E2 23052.907} C_VEL
LIN {X 0,Y 505.788,Z 351.206,A -85,B 0,C 180,E1 23049.559,E2 23049.559} C_VEL
LIN {X 0,Y 505.789,Z 351.207,A -85,B 0,C 180,E1 23046.014,E2 23046.014} C_VEL
LIN {X 0,Y 505.844,Z 351.201,A -85,B 0,C 180,E1 23042.719,E2 23042.719} C_VEL
LIN {X 0,Y 505.786,Z 351.209,A -85,B 0,C 180,E1 23039.434,E2 23039.434} C_VEL
LIN {X 0,Y 505.8,Z 351.206,A -85,B 0,C 180,E1 23035.919,E2 23035.919} C_VEL
LIN {X 0,Y 505.834,Z 351.206,A -85,B 0,C 180,E1 23032.618,E2 23032.618} C_VEL
LIN {X 0,Y 505.786,Z 351.191,A -85,B 0,C 180,E1 23029.261,E2 23029.261} C_VEL
LIN {X 0,Y 505.812,Z 351.156,A -85,B 0,C 180,E1 23025.811,E2 23025.811} C_VEL
LIN {X 0,Y 505.881,Z 351.386,A -85,B 0,C 180,E1 23024.112,E2 23024.112} C_VEL
LIN {X 0,Y 506.787,Z 354.164,A -85,B 0,C 180,E1 23023.7,E2 23023.7} C_VEL
LIN {X 0,Y 509.113,Z 356.733,A -85,B 0,C 180,E1 23022.866,E2 23022.866} C_VEL
LIN {X 0,Y 511.606,Z 358.017,A -85,B 0,C 180,E1 23022.072,E2 23022.072} C_VEL
LIN {X 0,Y 513.391,Z 361.447,A -85,B 0,C 180,E1 23021.432,E2 23021.432} C_VEL
LIN {X 0,Y 516.301,Z 363.937,A -85,B 0,C 180,E1 23020.543,E2 23020.543} C_VEL
LIN {X 0,Y 517.359,Z 364.778,A -85,B 0,C 180,E1 23020.231,E2 23020.231} C_VEL
LIN {X 0,Y 519.693,Z 368.414,A -85,B 0,C 180,E1 23019.502,E2 23019.502} C_VEL
LIN {X 0,Y 522.918,Z 371.268,A -85,B 0,C 180,E1 23018.608,E2 23018.608} C_VEL
LIN {X 0,Y 525.914,Z 375.327,A -85,B 0,C 180,E1 23017.769,E2 23017.769} C_VEL
LIN {X 0,Y 528.347,Z 377.593,A -85,B 0,C 180,E1 23017.143,E2 23017.143} C_VEL
LIN {X 0,Y 531.732,Z 381.856,A -85,B 0,C 180,E1 23016.271,E2 23016.271} C_VEL
LIN {X 0,Y 533.644,Z 383.935,A -85,B 0,C 180,E1 23015.803,E2 23015.803} C_VEL
LIN {X 0,Y 542.09,Z 394.626,A -85,B 0,C 180,E1 23013.813,E2 23013.813} C_VEL
LIN {X 0,Y 553.154,Z 409.334,A -85,B 0,C 180,E1 23011.437,E2 23011.437} C_VEL
LIN {X 0,Y 564.162,Z 424.894,A -85,B 0,C 180,E1 23009.277,E2 23009.277} C_VEL
LIN {X 0,Y 575.125,Z 440.838,A -85,B 0,C 180,E1 23007.299,E2 23007.299} C_VEL
LIN {X 0,Y 583.708,Z 453.765,A -85,B 0,C 180,E1 23005.846,E2 23005.846} C_VEL
LIN {X 0,Y 575.132,Z 669.725,A -85,B 0,C 180,E1 23002.652,E2 23002.652} C_VEL
LIN {X 0,Y 569.047,Z 825.92,A -85,B 0,C 180,E1 23000.353,E2 23000.353} C_VEL
LIN {X 0,Y 567.169,Z 851.137,A -85,B 0,C 180,E1 22999.886,E2 22999.886} C_VEL
LIN {X 0,Y 564.244,Z 879.162,A -85,B 0,C 180,E1 22999.175,E2 22999.175} C_VEL
LIN {X 0,Y 561.505,Z 900.749,A -85,B 0,C 180,E1 22998.484,E2 22998.484} C_VEL
LIN {X 0,Y 558.64,Z 920.558,A -85,B 0,C 180,E1 22997.731,E2 22997.731} C_VEL
LIN {X 0,Y 555.337,Z 940.956,A -85,B 0,C 180,E1 22996.827,E2 22996.827} C_VEL
LIN {X 0,Y 551.535,Z 962.316,A -85,B 0,C 180,E1 22995.732,E2 22995.732} C_VEL
LIN {X 0,Y 546.361,Z 988.655,A -85,B 0,C 180,E1 22994.14,E2 22994.14} C_VEL
LIN {X 0,Y 542.127,Z 1008.496,A -85,B 0,C 180,E1 22992.743,E2 22992.743} C_VEL
LIN {X 0,Y 538.022,Z 1026.87,A -85,B 0,C 180,E1 22991.279,E2 22991.279} C_VEL
LIN {X 0,Y 533.859,Z 1044.899,A -85,B 0,C 180,E1 22989.665,E2 22989.665} C_VEL
LIN {X 0,Y 528.87,Z 1066.25,A -85,B 0,C 180,E1 22987.5,E2 22987.5} C_VEL
LIN {X 0,Y 524.592,Z 1084.157,A -85,B 0,C 180,E1 22985.409,E2 22985.409} C_VEL
LIN {X 0,Y 521,Z 1099.403,A -85,B 0,C 180,E1 22983.421,E2 22983.421} C_VEL
LIN {X 0,Y 517.816,Z 1113.289,A -85,B 0,C 180,E1 22981.406,E2 22981.406} C_VEL
LIN {X 0,Y 514.613,Z 1127.784,A -85,B 0,C 180,E1 22979.06,E2 22979.06} C_VEL
LIN {X 0,Y 511.359,Z 1143.687,A -85,B 0,C 180,E1 22976.1,E2 22976.1} C_VEL
LIN {X 0,Y 509.183,Z 1155.251,A -85,B 0,C 180,E1 22973.615,E2 22973.615} C_VEL
LIN {X 0,Y 507.544,Z 1164.974,A -85,B 0,C 180,E1 22971.252,E2 22971.252} C_VEL
LIN {X 0,Y 506.26,Z 1173.912,A -85,B 0,C 180,E1 22968.779,E2 22968.779} C_VEL
LIN {X 0,Y 505.112,Z 1183.63,A -85,B 0,C 180,E1 22965.617,E2 22965.617} C_VEL
LIN {X 0,Y 504.468,Z 1190.63,A -85,B 0,C 180,E1 22962.791,E2 22962.791} C_VEL
LIN {X 0,Y 504.156,Z 1195.69,A -85,B 0,C 180,E1 22960.282,E2 22960.282} C_VEL
LIN {X 0,Y 504.002,Z 1199.515,A -85,B 0,C 180,E1 22957.868,E2 22957.868} C_VEL
LIN {X 0,Y 503.932,Z 1202.424,A -85,B 0,C 180,E1 22955.351,E2 22955.351} C_VEL
LIN {X 0,Y 503.91,Z 1204.438,A -85,B 0,C 180,E1 22952.502,E2 22952.502} C_VEL
LIN {X 0,Y 503.895,Z 1204.894,A -85,B 0,C 180,E1 22949.432,E2 22949.432} C_VEL
LIN {X 0,Y 503.916,Z 1204.029,A -85,B 0,C 180,E1 22946.815,E2 22946.815} C_VEL
LIN {X 0,Y 503.935,Z 1202.196,A -85,B 0,C 180,E1 22944.421,E2 22944.421} C_VEL
LIN {X 0,Y 504.008,Z 1199.354,A -85,B 0,C 180,E1 22942.018,E2 22942.018} C_VEL
LIN {X 0,Y 504.167,Z 1195.483,A -85,B 0,C 180,E1 22939.603,E2 22939.603} C_VEL
LIN {X 0,Y 504.523,Z 1190.047,A -85,B 0,C 180,E1 22936.943,E2 22936.943} C_VEL
LIN {X 0,Y 505.268,Z 1181.973,A -85,B 0,C 180,E1 22933.798,E2 22933.798} C_VEL
LIN {X 0,Y 506.326,Z 1173.402,A -85,B 0,C 180,E1 22931.073,E2 22931.073} C_VEL
LIN {X 0,Y 507.614,Z 1164.519,A -85,B 0,C 180,E1 22928.63,E2 22928.63} C_VEL
LIN {X 0,Y 509.278,Z 1154.743,A -85,B 0,C 180,E1 22926.267,E2 22926.267} C_VEL
LIN {X 0,Y 511.858,Z 1141.399,A -85,B 0,C 180,E1 22923.428,E2 22923.428} C_VEL
LIN {X 0,Y 514.953,Z 1126.183,A -85,B 0,C 180,E1 22920.672,E2 22920.672} C_VEL
LIN {X 0,Y 517.837,Z 1113.174,A -85,B 0,C 180,E1 22918.579,E2 22918.579} C_VEL
LIN {X 0,Y 520.998,Z 1099.377,A -85,B 0,C 180,E1 22916.579,E2 22916.579} C_VEL
LIN {X 0,Y 524.586,Z 1084.121,A -85,B 0,C 180,E1 22914.59,E2 22914.59} C_VEL
LIN {X 0,Y 529.354,Z 1064.065,A -85,B 0,C 180,E1 22912.267,E2 22912.267} C_VEL
LIN {X 0,Y 534.011,Z 1044.11,A -85,B 0,C 180,E1 22910.267,E2 22910.267} C_VEL
LIN {X 0,Y 538.248,Z 1025.79,A -85,B 0,C 180,E1 22908.634,E2 22908.634} C_VEL
LIN {X 0,Y 542.813,Z 1005.621,A -85,B 0,C 180,E1 22907.036,E2 22907.036} C_VEL
LIN {X 0,Y 548.176,Z 980.693,A -85,B 0,C 180,E1 22905.328,E2 22905.328} C_VEL
LIN {X 0,Y 552.228,Z 960.249,A -85,B 0,C 180,E1 22904.119,E2 22904.119} C_VEL
LIN {X 0,Y 555.893,Z 940.386,A -85,B 0,C 180,E1 22903.093,E2 22903.093} C_VEL
LIN {X 0,Y 559.321,Z 920.135,A -85,B 0,C 180,E1 22902.186,E2 22902.186} C_VEL
LIN {X 0,Y 562.564,Z 898.761,A -85,B 0,C 180,E1 22901.369,E2 22901.369} C_VEL
LIN {X 0,Y 566.044,Z 872.367,A -85,B 0,C 180,E1 22900.541,E2 22900.541} C_VEL
LIN {X 0,Y 568.661,Z 846.517,A -85,B 0,C 180,E1 22899.923,E2 22899.923} C_VEL
LIN {X 0,Y 570.374,Z 824.114,A -85,B 0,C 180,E1 22899.513,E2 22899.513} C_VEL
LIN {X 0,Y 579.804,Z 608.997,A -85,B 0,C 180,E1 22896.282,E2 22896.282} C_VEL
LIN {X 0,Y 586.924,Z 453.923,A -85,B 0,C 180,E1 22893.919,E2 22893.919} C_VEL
LIN {X 0,Y 578.329,Z 440.174,A -85,B 0,C 180,E1 22892.175,E2 22892.175} C_VEL
LIN {X 0,Y 568.14,Z 425.424,A -85,B 0,C 180,E1 22889.93,E2 22889.93} C_VEL
LIN {X 0,Y 560.844,Z 415.474,A -85,B 0,C 180,E1 22888.165,E2 22888.165} C_VEL
LIN {X 0,Y 556.684,Z 410.032,A -85,B 0,C 180,E1 22887.086,E2 22887.086} C_VEL
LIN {X 0,Y 552.801,Z 404.862,A -85,B 0,C 180,E1 22886.016,E2 22886.016} C_VEL
LIN {X 0,Y 548.59,Z 399.422,A -85,B 0,C 180,E1 22884.785,E2 22884.785} C_VEL
LIN {X 0,Y 545.043,Z 395.21,A -85,B 0,C 180,E1 22883.688,E2 22883.688} C_VEL
LIN {X 0,Y 541.412,Z 390.561,A -85,B 0,C 180,E1 22882.476,E2 22882.476} C_VEL
LIN {X 0,Y 538.063,Z 387.114,A -85,B 0,C 180,E1 22881.303,E2 22881.303} C_VEL
LIN {X 0,Y 536.341,Z 384.57,A -85,B 0,C 180,E1 22880.631,E2 22880.631} C_VEL
LIN {X 0,Y 533.013,Z 381.649,A -85,B 0,C 180,E1 22879.336,E2 22879.336} C_VEL
LIN {X 0,Y 531.073,Z 378.33,A -85,B 0,C 180,E1 22878.44,E2 22878.44} C_VEL
LIN {X 0,Y 527.367,Z 375.566,A -85,B 0,C 180,E1 22876.75,E2 22876.75} C_VEL
LIN {X 0,Y 525.394,Z 372.117,A -85,B 0,C 180,E1 22875.622,E2 22875.622} C_VEL
LIN {X 0,Y 524.711,Z 371.575,A -85,B 0,C 180,E1 22875.247,E2 22875.247} C_VEL
LIN {X 0,Y 521.645,Z 369.523,A -85,B 0,C 180,E1 22873.411,E2 22873.411} C_VEL
LIN {X 0,Y 519.701,Z 366.541,A -85,B 0,C 180,E1 22871.88,E2 22871.88} C_VEL
LIN {X 0,Y 519.158,Z 364.97,A -85,B 0,C 180,E1 22871.33,E2 22871.33} C_VEL
LIN {X 0,Y 514.489,Z 362.212,A -85,B 0,C 180,E1 22864.347,E2 22864.347} C_VEL
LIN {X 0,Y 514.776,Z 362.437,A -85,B 0,C 180,E1 22861.224,E2 22861.224} C_VEL
LIN {X 0,Y 519.274,Z 365.119,A -85,B 0,C 180,E1 22855.361,E2 22855.361} C_VEL
LIN {X 0,Y 520.58,Z 368.27,A -85,B 0,C 180,E1 22854.157,E2 22854.157} C_VEL
LIN {X 0,Y 523.709,Z 371.12,A -85,B 0,C 180,E1 22852.099,E2 22852.099} C_VEL
LIN {X 0,Y 525.332,Z 371.929,A -85,B 0,C 180,E1 22851.214,E2 22851.214} C_VEL
LIN {X 0,Y 527.227,Z 375.393,A -85,B 0,C 180,E1 22850.117,E2 22850.117} C_VEL
LIN {X 0,Y 530.764,Z 378.219,A -85,B 0,C 180,E1 22848.481,E2 22848.481} C_VEL
LIN {X 0,Y 531.462,Z 379.072,A -85,B 0,C 180,E1 22848.166,E2 22848.166} C_VEL
LIN {X 0,Y 534.084,Z 382.839,A -85,B 0,C 180,E1 22847.017,E2 22847.017} C_VEL
LIN {X 0,Y 536.938,Z 385.259,A -85,B 0,C 180,E1 22845.935,E2 22845.935} C_VEL
LIN {X 0,Y 539.946,Z 389.345,A -85,B 0,C 180,E1 22844.809,E2 22844.809} C_VEL
LIN {X 0,Y 542.286,Z 391.479,A -85,B 0,C 180,E1 22844.026,E2 22844.026} C_VEL
LIN {X 0,Y 545.72,Z 395.839,A -85,B 0,C 180,E1 22842.898,E2 22842.898} C_VEL
LIN {X 0,Y 547.59,Z 397.771,A -85,B 0,C 180,E1 22842.328,E2 22842.328} C_VEL
LIN {X 0,Y 551.506,Z 402.438,A -85,B 0,C 180,E1 22841.173,E2 22841.173} C_VEL
LIN {X 0,Y 557.96,Z 410.435,A -85,B 0,C 180,E1 22839.409,E2 22839.409} C_VEL
LIN {X 0,Y 562.265,Z 415.842,A -85,B 0,C 180,E1 22838.318,E2 22838.318} C_VEL
LIN {X 0,Y 569.774,Z 425.37,A -85,B 0,C 180,E1 22836.552,E2 22836.552} C_VEL
LIN {X 0,Y 578.087,Z 437.174,A -85,B 0,C 180,E1 22834.736,E2 22834.736} C_VEL
LIN {X 0,Y 586.942,Z 450.843,A -85,B 0,C 180,E1 22832.945,E2 22832.945} C_VEL
LIN {X 0,Y 577.627,Z 653.651,A -85,B 0,C 180,E1 22829.869,E2 22829.869} C_VEL
LIN {X 0,Y 570.376,Z 818.349,A -85,B 0,C 180,E1 22827.393,E2 22827.393} C_VEL
LIN {X 0,Y 568.355,Z 843.973,A -85,B 0,C 180,E1 22826.905,E2 22826.905} C_VEL
LIN {X 0,Y 565.319,Z 871.353,A -85,B 0,C 180,E1 22826.192,E2 22826.192} C_VEL
LIN {X 0,Y 562.434,Z 892.943,A -85,B 0,C 180,E1 22825.485,E2 22825.485} C_VEL
LIN {X 0,Y 559.336,Z 913.324,A -85,B 0,C 180,E1 22824.689,E2 22824.689} C_VEL
LIN {X 0,Y 555.893,Z 933.486,A -85,B 0,C 180,E1 22823.774,E2 22823.774} C_VEL
LIN {X 0,Y 551.399,Z 957.634,A -85,B 0,C 180,E1 22822.497,E2 22822.497} C_VEL
LIN {X 0,Y 546.388,Z 981.666,A -85,B 0,C 180,E1 22820.985,E2 22820.985} C_VEL
LIN {X 0,Y 542.17,Z 1000.773,A -85,B 0,C 180,E1 22819.609,E2 22819.609} C_VEL
LIN {X 0,Y 539.884,Z 1011.139,A -85,B 0,C 180,E1 22818.797,E2 22818.797} C_VEL
LIN {X 0,Y 537.619,Z 1017.404,A -85,B 0,C 180,E1 22818.348,E2 22818.348} C_VEL
LIN {X 0,Y 529.125,Z 1033.25,A -85,B 0,C 180,E1 22817.375,E2 22817.375} C_VEL
LIN {X 0,Y 526.935,Z 1039.045,A -85,B 0,C 180,E1 22816.89,E2 22816.89} C_VEL
LIN {X 0,Y 521.677,Z 1059.955,A -85,B 0,C 180,E1 22814.676,E2 22814.676} C_VEL
LIN {X 0,Y 517.253,Z 1077.467,A -85,B 0,C 180,E1 22812.565,E2 22812.565} C_VEL
LIN {X 0,Y 512.901,Z 1094.931,A -85,B 0,C 180,E1 22810.185,E2 22810.185} C_VEL
LIN {X 0,Y 508.622,Z 1112.672,A -85,B 0,C 180,E1 22807.404,E2 22807.404} C_VEL
LIN {X 0,Y 505.09,Z 1128.026,A -85,B 0,C 180,E1 22804.62,E2 22804.62} C_VEL
LIN {X 0,Y 502.524,Z 1140.247,A -85,B 0,C 180,E1 22802.089,E2 22802.089} C_VEL
LIN {X 0,Y 500.158,Z 1153.106,A -85,B 0,C 180,E1 22799.063,E2 22799.063} C_VEL
LIN {X 0,Y 498.487,Z 1163.427,A -85,B 0,C 180,E1 22796.185,E2 22796.185} C_VEL
LIN {X 0,Y 497.43,Z 1171.478,A -85,B 0,C 180,E1 22793.578,E2 22793.578} C_VEL
LIN {X 0,Y 496.682,Z 1178.872,A -85,B 0,C 180,E1 22790.751,E2 22790.751} C_VEL
LIN {X 0,Y 496.191,Z 1185.375,A -85,B 0,C 180,E1 22787.593,E2 22787.593} C_VEL
LIN {X 0,Y 496.016,Z 1189.512,A -85,B 0,C 180,E1 22784.953,E2 22784.953} C_VEL
LIN {X 0,Y 495.937,Z 1192.355,A -85,B 0,C 180,E1 22782.458,E2 22782.458} C_VEL
LIN {X 0,Y 495.914,Z 1194.213,A -85,B 0,C 180,E1 22779.868,E2 22779.868} C_VEL
LIN {X 0,Y 495.91,Z 1194.983,A -85,B 0,C 180,E1 22776.832,E2 22776.832} C_VEL
LIN {X 0,Y 495.908,Z 1194.15,A -85,B 0,C 180,E1 22773.931,E2 22773.931} C_VEL
LIN {X 0,Y 495.931,Z 1192.294,A -85,B 0,C 180,E1 22771.386,E2 22771.386} C_VEL
LIN {X 0,Y 496.014,Z 1189.363,A -85,B 0,C 180,E1 22768.845,E2 22768.845} C_VEL
LIN {X 0,Y 496.208,Z 1184.956,A -85,B 0,C 180,E1 22766.072,E2 22766.072} C_VEL
LIN {X 0,Y 496.744,Z 1178.055,A -85,B 0,C 180,E1 22762.831,E2 22762.831} C_VEL
LIN {X 0,Y 497.497,Z 1170.995,A -85,B 0,C 180,E1 22760.164,E2 22760.164} C_VEL
LIN {X 0,Y 498.561,Z 1163.044,A -85,B 0,C 180,E1 22757.609,E2 22757.609} C_VEL
LIN {X 0,Y 500.33,Z 1152.073,A -85,B 0,C 180,E1 22754.586,E2 22754.586} C_VEL
LIN {X 0,Y 502.637,Z 1139.605,A -85,B 0,C 180,E1 22751.682,E2 22751.682} C_VEL
LIN {X 0,Y 505.268,Z 1127.218,A -85,B 0,C 180,E1 22749.133,E2 22749.133} C_VEL
LIN {X 0,Y 509.112,Z 1110.44,A -85,B 0,C 180,E1 22746.136,E2 22746.136} C_VEL
LIN {X 0,Y 513.273,Z 1093.409,A -85,B 0,C 180,E1 22743.507,E2 22743.507} C_VEL
LIN {X 0,Y 517.951,Z 1074.644,A -85,B 0,C 180,E1 22740.987,E2 22740.987} C_VEL
LIN {X 0,Y 523.204,Z 1053.836,A -85,B 0,C 180,E1 22738.553,E2 22738.553} C_VEL
LIN {X 0,Y 527.82,Z 1035.194,A -85,B 0,C 180,E1 22736.66,E2 22736.66} C_VEL
LIN {X 0,Y 532.026,Z 1017.836,A -85,B 0,C 180,E1 22735.092,E2 22735.092} C_VEL
LIN {X 0,Y 536.247,Z 999.712,A -85,B 0,C 180,E1 22733.635,E2 22733.635} C_VEL
LIN {X 0,Y 541.282,Z 977.105,A -85,B 0,C 180,E1 22732.04,E2 22732.04} C_VEL
LIN {X 0,Y 546.149,Z 952.839,A -85,B 0,C 180,E1 22730.588,E2 22730.588} C_VEL
LIN {X 0,Y 549.925,Z 932.262,A -85,B 0,C 180,E1 22729.527,E2 22729.527} C_VEL
LIN {X 0,Y 553.204,Z 912.685,A -85,B 0,C 180,E1 22728.654,E2 22728.654} C_VEL
LIN {X 0,Y 556.383,Z 891.349,A -85,B 0,C 180,E1 22727.84,E2 22727.84} C_VEL
LIN {X 0,Y 559.723,Z 865.437,A -85,B 0,C 180,E1 22727.023,E2 22727.023} C_VEL
LIN {X 0,Y 562.331,Z 838.718,A -85,B 0,C 180,E1 22726.383,E2 22726.383} C_VEL
LIN {X 0,Y 563.987,Z 816.201,A -85,B 0,C 180,E1 22725.975,E2 22725.975} C_VEL
LIN {X 0,Y 572.156,Z 614.039,A -85,B 0,C 180,E1 22722.985,E2 22722.985} C_VEL
LIN {X 0,Y 578.776,Z 454.621,A -85,B 0,C 180,E1 22720.608,E2 22720.608} C_VEL
LIN {X 0,Y 561.985,Z 430.216,A -85,B 0,C 180,E1 22717.609,E2 22717.609} C_VEL
LIN {X 0,Y 551.269,Z 416.177,A -85,B 0,C 180,E1 22715.512,E2 22715.512} C_VEL
LIN {X 0,Y 542.667,Z 405.262,A -85,B 0,C 180,E1 22713.684,E2 22713.684} C_VEL
LIN {X 0,Y 538.479,Z 400.097,A -85,B 0,C 180,E1 22712.74,E2 22712.74} C_VEL
LIN {X 0,Y 534.21,Z 394.822,A -85,B 0,C 180,E1 22711.733,E2 22711.733} C_VEL
LIN {X 0,Y 529.781,Z 389.441,A -85,B 0,C 180,E1 22710.637,E2 22710.637} C_VEL
LIN {X 0,Y 526.005,Z 384.743,A -85,B 0,C 180,E1 22709.651,E2 22709.651} C_VEL
LIN {X 0,Y 521.745,Z 380.171,A -85,B 0,C 180,E1 22708.502,E2 22708.502} C_VEL
LIN {X 0,Y 520.144,Z 377.936,A -85,B 0,C 180,E1 22708.035,E2 22708.035} C_VEL
LIN {X 0,Y 516.723,Z 374.567,A -85,B 0,C 180,E1 22707.048,E2 22707.048} C_VEL
LIN {X 0,Y 514.929,Z 371.815,A -85,B 0,C 180,E1 22706.474,E2 22706.474} C_VEL
LIN {X 0,Y 511.645,Z 369.092,A -85,B 0,C 180,E1 22705.464,E2 22705.464} C_VEL
LIN {X 0,Y 509.519,Z 365.547,A -85,B 0,C 180,E1 22704.708,E2 22704.708} C_VEL
LIN {X 0,Y 506.31,Z 363.363,A -85,B 0,C 180,E1 22703.634,E2 22703.634} C_VEL
LIN {X 0,Y 504.284,Z 360.115,A -85,B 0,C 180,E1 22702.838,E2 22702.838} C_VEL
LIN {X 0,Y 503.853,Z 358.928,A -85,B 0,C 180,E1 22702.643,E2 22702.643} C_VEL
LIN {X 0,Y 500.482,Z 357.103,A -85,B 0,C 180,E1 22701.384,E2 22701.384} C_VEL
LIN {X 0,Y 498.424,Z 354.294,A -85,B 0,C 180,E1 22700.476,E2 22700.476} C_VEL
LIN {X 0,Y 497.837,Z 352.155,A -85,B 0,C 180,E1 22700.087,E2 22700.087} C_VEL
LIN {X 0,Y 497.876,Z 352.193,A -85,B 0,C 180,E1 22696.679,E2 22696.679} C_VEL
LIN {X 0,Y 497.859,Z 352.195,A -85,B 0,C 180,E1 22693.472,E2 22693.472} C_VEL
LIN {X 0,Y 497.845,Z 352.195,A -85,B 0,C 180,E1 22689.946,E2 22689.946} C_VEL
LIN {X 0,Y 497.896,Z 352.19,A -85,B 0,C 180,E1 22686.573,E2 22686.573} C_VEL
LIN {X 0,Y 497.861,Z 352.198,A -85,B 0,C 180,E1 22683.224,E2 22683.224} C_VEL
LIN {X 0,Y 497.848,Z 352.201,A -85,B 0,C 180,E1 22679.77,E2 22679.77} C_VEL
LIN {X 0,Y 497.905,Z 352.196,A -85,B 0,C 180,E1 22676.409,E2 22676.409} C_VEL
LIN {X 0,Y 497.858,Z 352.206,A -85,B 0,C 180,E1 22673.079,E2 22673.079} C_VEL
LIN {X 0,Y 497.855,Z 352.19,A -85,B 0,C 180,E1 22669.586,E2 22669.586} C_VEL
LIN {X 0,Y 497.873,Z 352.306,A -85,B 0,C 180,E1 22666.942,E2 22666.942} C_VEL
LIN {X 0,Y 498.768,Z 354.907,A -85,B 0,C 180,E1 22666.464,E2 22666.464} C_VEL
LIN {X 0,Y 501.177,Z 357.708,A -85,B 0,C 180,E1 22665.441,E2 22665.441} C_VEL
LIN {X 0,Y 503.905,Z 359.155,A -85,B 0,C 180,E1 22664.432,E2 22664.432} C_VEL
LIN {X 0,Y 505.554,Z 362.48,A -85,B 0,C 180,E1 22663.748,E2 22663.748} C_VEL
LIN {X 0,Y 508.486,Z 365.008,A -85,B 0,C 180,E1 22662.727,E2 22662.727} C_VEL
LIN {X 0,Y 509.712,Z 365.798,A -85,B 0,C 180,E1 22662.328,E2 22662.328} C_VEL
LIN {X 0,Y 511.912,Z 369.372,A -85,B 0,C 180,E1 22661.553,E2 22661.553} C_VEL
LIN {X 0,Y 515.332,Z 372.281,A -85,B 0,C 180,E1 22660.505,E2 22660.505} C_VEL
LIN {X 0,Y 518.183,Z 376.32,A -85,B 0,C 180,E1 22659.617,E2 22659.617} C_VEL
LIN {X 0,Y 520.914,Z 378.88,A -85,B 0,C 180,E1 22658.847,E2 22658.847} C_VEL
LIN {X 0,Y 524.185,Z 383.038,A -85,B 0,C 180,E1 22657.927,E2 22657.927} C_VEL
LIN {X 0,Y 526.202,Z 385.04,A -85,B 0,C 180,E1 22657.399,E2 22657.399} C_VEL
LIN {X 0,Y 529.966,Z 389.572,A -85,B 0,C 180,E1 22656.423,E2 22656.423} C_VEL
LIN {X 0,Y 538.682,Z 400.433,A -85,B 0,C 180,E1 22654.315,E2 22654.315} C_VEL
LIN {X 0,Y 550.566,Z 416.529,A -85,B 0,C 180,E1 22651.705,E2 22651.705} C_VEL
LIN {X 0,Y 562.557,Z 433.584,A -85,B 0,C 180,E1 22649.328,E2 22649.328} C_VEL
LIN {X 0,Y 577.998,Z 456.486,A -85,B 0,C 180,E1 22646.566,E2 22646.566} C_VEL
LIN {X 0,Y 578.802,Z 458.123,A -85,B 0,C 180,E1 22646.421,E2 22646.421} C_VEL
LIN {X 0,Y 569.873,Z 674.795,A -85,B 0,C 180,E1 22643.201,E2 22643.201} C_VEL
LIN {X 0,Y 563.773,Z 825.885,A -85,B 0,C 180,E1 22640.965,E2 22640.965} C_VEL
LIN {X 0,Y 561.823,Z 851.325,A -85,B 0,C 180,E1 22640.492,E2 22640.492} C_VEL
LIN {X 0,Y 558.804,Z 879.311,A -85,B 0,C 180,E1 22639.779,E2 22639.779} C_VEL
LIN {X 0,Y 556.004,Z 900.717,A -85,B 0,C 180,E1 22639.092,E2 22639.092} C_VEL
LIN {X 0,Y 552.952,Z 921.122,A -85,B 0,C 180,E1 22638.313,E2 22638.313} C_VEL
LIN {X 0,Y 549.524,Z 941.593,A -85,B 0,C 180,E1 22637.4,E2 22637.4} C_VEL
LIN {X 0,Y 545.042,Z 965.958,A -85,B 0,C 180,E1 22636.132,E2 22636.132} C_VEL
LIN {X 0,Y 540.048,Z 990.072,A -85,B 0,C 180,E1 22634.637,E2 22634.637} C_VEL
LIN {X 0,Y 535.943,Z 1008.702,A -85,B 0,C 180,E1 22633.313,E2 22633.313} C_VEL
LIN {X 0,Y 531.784,Z 1026.709,A -85,B 0,C 180,E1 22631.872,E2 22631.872} C_VEL
LIN {X 0,Y 527.509,Z 1044.557,A -85,B 0,C 180,E1 22630.266,E2 22630.266} C_VEL
LIN {X 0,Y 522.489,Z 1065.117,A -85,B 0,C 180,E1 22628.178,E2 22628.178} C_VEL
LIN {X 0,Y 517.634,Z 1084.521,A -85,B 0,C 180,E1 22625.89,E2 22625.89} C_VEL
LIN {X 0,Y 513.984,Z 1099.302,A -85,B 0,C 180,E1 22623.938,E2 22623.938} C_VEL
LIN {X 0,Y 510.673,Z 1113.092,A -85,B 0,C 180,E1 22621.913,E2 22621.913} C_VEL
LIN {X 0,Y 507.44,Z 1126.982,A -85,B 0,C 180,E1 22619.641,E2 22619.641} C_VEL
LIN {X 0,Y 503.845,Z 1143.617,A -85,B 0,C 180,E1 22616.519,E2 22616.519} C_VEL
LIN {X 0,Y 501.607,Z 1154.889,A -85,B 0,C 180,E1 22614.081,E2 22614.081} C_VEL
LIN {X 0,Y 499.878,Z 1164.513,A -85,B 0,C 180,E1 22611.718,E2 22611.718} C_VEL
LIN {X 0,Y 498.544,Z 1173.101,A -85,B 0,C 180,E1 22609.324,E2 22609.324} C_VEL
LIN {X 0,Y 497.417,Z 1181.622,A -85,B 0,C 180,E1 22606.585,E2 22606.585} C_VEL
LIN {X 0,Y 496.6,Z 1189.79,A -85,B 0,C 180,E1 22603.388,E2 22603.388} C_VEL
LIN {X 0,Y 496.197,Z 1195.274,A -85,B 0,C 180,E1 22600.683,E2 22600.683} C_VEL
LIN {X 0,Y 496.018,Z 1199.233,A -85,B 0,C 180,E1 22598.199,E2 22598.199} C_VEL
LIN {X 0,Y 495.94,Z 1202.081,A -85,B 0,C 180,E1 22595.785,E2 22595.785} C_VEL
LIN {X 0,Y 495.915,Z 1203.959,A -85,B 0,C 180,E1 22593.352,E2 22593.352} C_VEL
LIN {X 0,Y 495.906,Z 1204.826,A -85,B 0,C 180,E1 22590.924,E2 22590.924} C_VEL
LIN {X 0,Y 495.91,Z 1204.712,A -85,B 0,C 180,E1 22588.498,E2 22588.498} C_VEL
LIN {X 0,Y 495.919,Z 1203.413,A -85,B 0,C 180,E1 22585.722,E2 22585.722} C_VEL
LIN {X 0,Y 495.988,Z 1200.309,A -85,B 0,C 180,E1 22582.587,E2 22582.587} C_VEL
LIN {X 0,Y 496.144,Z 1196.306,A -85,B 0,C 180,E1 22579.902,E2 22579.902} C_VEL
LIN {X 0,Y 496.455,Z 1191.316,A -85,B 0,C 180,E1 22577.319,E2 22577.319} C_VEL
LIN {X 0,Y 497.003,Z 1185.444,A -85,B 0,C 180,E1 22574.839,E2 22574.839} C_VEL
LIN {X 0,Y 497.898,Z 1177.734,A -85,B 0,C 180,E1 22572.107,E2 22572.107} C_VEL
LIN {X 0,Y 499.522,Z 1166.783,A -85,B 0,C 180,E1 22568.875,E2 22568.875} C_VEL
LIN {X 0,Y 501.326,Z 1156.414,A -85,B 0,C 180,E1 22566.273,E2 22566.273} C_VEL
LIN {X 0,Y 503.235,Z 1146.506,A -85,B 0,C 180,E1 22564.08,E2 22564.08} C_VEL
LIN {X 0,Y 505.673,Z 1134.942,A -85,B 0,C 180,E1 22561.799,E2 22561.799} C_VEL
LIN {X 0,Y 508.726,Z 1121.322,A -85,B 0,C 180,E1 22559.4,E2 22559.4} C_VEL
LIN {X 0,Y 513.171,Z 1102.669,A -85,B 0,C 180,E1 22556.537,E2 22556.537} C_VEL
LIN {X 0,Y 516.94,Z 1087.268,A -85,B 0,C 180,E1 22554.464,E2 22554.464} C_VEL
LIN {X 0,Y 520.668,Z 1072.2,A -85,B 0,C 180,E1 22552.64,E2 22552.64} C_VEL
LIN {X 0,Y 524.657,Z 1056.135,A -85,B 0,C 180,E1 22550.891,E2 22550.891} C_VEL
LIN {X 0,Y 529.645,Z 1036,A -85,B 0,C 180,E1 22548.932,E2 22548.932} C_VEL
LIN {X 0,Y 535.092,Z 1013.032,A -85,B 0,C 180,E1 22546.998,E2 22546.998} C_VEL
LIN {X 0,Y 539.629,Z 993.252,A -85,B 0,C 180,E1 22545.542,E2 22545.542} C_VEL
LIN {X 0,Y 543.712,Z 974.573,A -85,B 0,C 180,E1 22544.328,E2 22544.328} C_VEL
LIN {X 0,Y 547.605,Z 955.571,A -85,B 0,C 180,E1 22543.237,E2 22543.237} C_VEL
LIN {X 0,Y 552.077,Z 931.828,A -85,B 0,C 180,E1 22542.052,E2 22542.052} C_VEL
LIN {X 0,Y 556.32,Z 905.926,A -85,B 0,C 180,E1 22540.988,E2 22540.988} C_VEL
LIN {X 0,Y 559.446,Z 884.082,A -85,B 0,C 180,E1 22540.248,E2 22540.248} C_VEL
LIN {X 0,Y 562.025,Z 862.903,A -85,B 0,C 180,E1 22539.656,E2 22539.656} C_VEL
LIN {X 0,Y 564.196,Z 841.283,A -85,B 0,C 180,E1 22539.175,E2 22539.175} C_VEL
LIN {X 0,Y 566.125,Z 813.662,A -85,B 0,C 180,E1 22538.7,E2 22538.7} C_VEL
LIN {X 0,Y 576.251,Z 589.271,A -85,B 0,C 180,E1 22535.322,E2 22535.322} C_VEL
LIN {X 0,Y 582.487,Z 458.106,A -85,B 0,C 180,E1 22533.304,E2 22533.304} C_VEL
LIN {X 0,Y 573.416,Z 443.709,A -85,B 0,C 180,E1 22531.396,E2 22531.396} C_VEL
LIN {X 0,Y 562.46,Z 427.817,A -85,B 0,C 180,E1 22528.859,E2 22528.859} C_VEL
LIN {X 0,Y 554.819,Z 417.643,A -85,B 0,C 180,E1 22526.895,E2 22526.895} C_VEL
LIN {X 0,Y 550.373,Z 411.72,A -85,B 0,C 180,E1 22525.648,E2 22525.648} C_VEL
LIN {X 0,Y 546.483,Z 406.611,A -85,B 0,C 180,E1 22524.483,E2 22524.483} C_VEL
LIN {X 0,Y 542.678,Z 402.075,A -85,B 0,C 180,E1 22523.28,E2 22523.28} C_VEL
LIN {X 0,Y 539.713,Z 398.15,A -85,B 0,C 180,E1 22522.263,E2 22522.263} C_VEL
LIN {X 0,Y 536.143,Z 394.296,A -85,B 0,C 180,E1 22520.982,E2 22520.982} C_VEL
LIN {X 0,Y 534.843,Z 392.296,A -85,B 0,C 180,E1 22520.463,E2 22520.463} C_VEL
LIN {X 0,Y 531.435,Z 389.207,A -85,B 0,C 180,E1 22519.11,E2 22519.11} C_VEL
LIN {X 0,Y 529.386,Z 385.982,A -85,B 0,C 180,E1 22518.159,E2 22518.159} C_VEL
LIN {X 0,Y 525.684,Z 382.887,A -85,B 0,C 180,E1 22516.407,E2 22516.407} C_VEL
LIN {X 0,Y 523.764,Z 379.536,A -85,B 0,C 180,E1 22515.275,E2 22515.275} C_VEL
LIN {X 0,Y 520.68,Z 377.579,A -85,B 0,C 180,E1 22513.436,E2 22513.436} C_VEL
LIN {X 0,Y 518.586,Z 374.536,A -85,B 0,C 180,E1 22511.793,E2 22511.793} C_VEL
LIN {X 0,Y 517.924,Z 372.866,A -85,B 0,C 180,E1 22511.131,E2 22511.131} C_VEL
LIN {X 0,Y 513.512,Z 370.154,A -85,B 0,C 180,E1 22504.355,E2 22504.355} C_VEL
LIN {X 0,Y 513.796,Z 370.384,A -85,B 0,C 180,E1 22501.227,E2 22501.227} C_VEL
LIN {X 0,Y 518.089,Z 373.029,A -85,B 0,C 180,E1 22495.517,E2 22495.517} C_VEL
LIN {X 0,Y 519.449,Z 376.16,A -85,B 0,C 180,E1 22494.255,E2 22494.255} C_VEL
LIN {X 0,Y 522.547,Z 378.995,A -85,B 0,C 180,E1 22492.192,E2 22492.192} C_VEL
LIN {X 0,Y 524.037,Z 379.908,A -85,B 0,C 180,E1 22491.358,E2 22491.358} C_VEL
LIN {X 0,Y 526.236,Z 383.549,A -85,B 0,C 180,E1 22490.098,E2 22490.098} C_VEL
LIN {X 0,Y 529.881,Z 386.623,A -85,B 0,C 180,E1 22488.406,E2 22488.406} C_VEL
LIN {X 0,Y 532.585,Z 390.509,A -85,B 0,C 180,E1 22487.201,E2 22487.201} C_VEL
LIN {X 0,Y 535.265,Z 392.833,A -85,B 0,C 180,E1 22486.166,E2 22486.166} C_VEL
LIN {X 0,Y 538.381,Z 397.016,A -85,B 0,C 180,E1 22484.984,E2 22484.984} C_VEL
LIN {X 0,Y 540.608,Z 399.18,A -85,B 0,C 180,E1 22484.223,E2 22484.223} C_VEL
LIN {X 0,Y 544.258,Z 403.661,A -85,B 0,C 180,E1 22483.016,E2 22483.016} C_VEL
LIN {X 0,Y 545.934,Z 405.596,A -85,B 0,C 180,E1 22482.493,E2 22482.493} C_VEL
LIN {X 0,Y 550.918,Z 411.664,A -85,B 0,C 180,E1 22481.014,E2 22481.014} C_VEL
LIN {X 0,Y 555.95,Z 417.902,A -85,B 0,C 180,E1 22479.634,E2 22479.634} C_VEL
LIN {X 0,Y 560.303,Z 423.455,A -85,B 0,C 180,E1 22478.513,E2 22478.513} C_VEL
LIN {X 0,Y 567.341,Z 432.492,A -85,B 0,C 180,E1 22476.83,E2 22476.83} C_VEL
LIN {X 0,Y 575.346,Z 444.023,A -85,B 0,C 180,E1 22475.047,E2 22475.047} C_VEL
LIN {X 0,Y 582.57,Z 455.289,A -85,B 0,C 180,E1 22473.545,E2 22473.545} C_VEL
LIN {X 0,Y 572.373,Z 668.776,A -85,B 0,C 180,E1 22470.299,E2 22470.299} C_VEL
LIN {X 0,Y 565.502,Z 818.493,A -85,B 0,C 180,E1 22468.036,E2 22468.036} C_VEL
LIN {X 0,Y 563.386,Z 844.403,A -85,B 0,C 180,E1 22467.54,E2 22467.54} C_VEL
LIN {X 0,Y 560.242,Z 871.663,A -85,B 0,C 180,E1 22466.826,E2 22466.826} C_VEL
LIN {X 0,Y 557.286,Z 893.047,A -85,B 0,C 180,E1 22466.124,E2 22466.124} C_VEL
LIN {X 0,Y 554.075,Z 913.383,A -85,B 0,C 180,E1 22465.328,E2 22465.328} C_VEL
LIN {X 0,Y 550.616,Z 932.916,A -85,B 0,C 180,E1 22464.441,E2 22464.441} C_VEL
LIN {X 0,Y 546.351,Z 954.959,A -85,B 0,C 180,E1 22463.28,E2 22463.28} C_VEL
LIN {X 0,Y 540.891,Z 980.484,A -85,B 0,C 180,E1 22461.693,E2 22461.693} C_VEL
LIN {X 0,Y 536.271,Z 1000.558,A -85,B 0,C 180,E1 22460.243,E2 22460.243} C_VEL
LIN {X 0,Y 531.905,Z 1018.778,A -85,B 0,C 180,E1 22458.756,E2 22458.756} C_VEL
LIN {X 0,Y 527.092,Z 1038.378,A -85,B 0,C 180,E1 22456.954,E2 22456.954} C_VEL
LIN {X 0,Y 526.935,Z 1039.045,A -85,B 0,C 180,E1 22456.89,E2 22456.89} C_VEL
LIN {X 0,Y 524.724,Z 1044.864,A -85,B 0,C 180,E1 22456.385,E2 22456.385} C_VEL
LIN {X 0,Y 516.017,Z 1059.651,A -85,B 0,C 180,E1 22455.219,E2 22455.219} C_VEL
LIN {X 0,Y 513.757,Z 1065.05,A -85,B 0,C 180,E1 22454.659,E2 22454.659} C_VEL
LIN {X 0,Y 508.852,Z 1083.79,A -85,B 0,C 180,E1 22452.298,E2 22452.298} C_VEL
LIN {X 0,Y 504.171,Z 1101.699,A -85,B 0,C 180,E1 22449.686,E2 22449.686} C_VEL
LIN {X 0,Y 500.316,Z 1117.186,A -85,B 0,C 180,E1 22447.116,E2 22447.116} C_VEL
LIN {X 0,Y 496.551,Z 1133.26,A -85,B 0,C 180,E1 22444.041,E2 22444.041} C_VEL
LIN {X 0,Y 493.613,Z 1146.955,A -85,B 0,C 180,E1 22440.964,E2 22440.964} C_VEL
LIN {X 0,Y 491.76,Z 1156.824,A -85,B 0,C 180,E1 22438.41,E2 22438.41} C_VEL
LIN {X 0,Y 490.316,Z 1165.883,A -85,B 0,C 180,E1 22435.744,E2 22435.744} C_VEL
LIN {X 0,Y 489.116,Z 1175.21,A -85,B 0,C 180,E1 22432.474,E2 22432.474} C_VEL
LIN {X 0,Y 488.479,Z 1181.546,A -85,B 0,C 180,E1 22429.739,E2 22429.739} C_VEL
LIN {X 0,Y 488.16,Z 1186.409,A -85,B 0,C 180,E1 22427.154,E2 22427.154} C_VEL
LIN {X 0,Y 487.994,Z 1190.307,A -85,B 0,C 180,E1 22424.476,E2 22424.476} C_VEL
LIN {X 0,Y 487.918,Z 1193.406,A -85,B 0,C 180,E1 22421.346,E2 22421.346} C_VEL
LIN {X 0,Y 487.912,Z 1194.719,A -85,B 0,C 180,E1 22418.485,E2 22418.485} C_VEL
LIN {X 0,Y 487.913,Z 1194.827,A -85,B 0,C 180,E1 22415.999,E2 22415.999} C_VEL
LIN {X 0,Y 487.911,Z 1193.947,A -85,B 0,C 180,E1 22413.525,E2 22413.525} C_VEL
LIN {X 0,Y 487.941,Z 1192.068,A -85,B 0,C 180,E1 22411.057,E2 22411.057} C_VEL
LIN {X 0,Y 488.04,Z 1188.896,A -85,B 0,C 180,E1 22408.356,E2 22408.356} C_VEL
LIN {X 0,Y 488.357,Z 1183.396,A -85,B 0,C 180,E1 22405.067,E2 22405.067} C_VEL
LIN {X 0,Y 488.855,Z 1177.474,A -85,B 0,C 180,E1 22402.36,E2 22402.36} C_VEL
LIN {X 0,Y 489.65,Z 1170.657,A -85,B 0,C 180,E1 22399.767,E2 22399.767} C_VEL
LIN {X 0,Y 490.861,Z 1162.278,A -85,B 0,C 180,E1 22397.052,E2 22397.052} C_VEL
LIN {X 0,Y 492.975,Z 1150.191,A -85,B 0,C 180,E1 22393.746,E2 22393.746} C_VEL
LIN {X 0,Y 495.312,Z 1138.646,A -85,B 0,C 180,E1 22391.034,E2 22391.034} C_VEL
LIN {X 0,Y 498.457,Z 1124.898,A -85,B 0,C 180,E1 22388.217,E2 22388.217} C_VEL
LIN {X 0,Y 502.462,Z 1108.421,A -85,B 0,C 180,E1 22385.299,E2 22385.299} C_VEL
LIN {X 0,Y 506.692,Z 1091.859,A -85,B 0,C 180,E1 22382.754,E2 22382.754} C_VEL
LIN {X 0,Y 511.125,Z 1074.926,A -85,B 0,C 180,E1 22380.465,E2 22380.465} C_VEL
LIN {X 0,Y 516.422,Z 1054.948,A -85,B 0,C 180,E1 22378.092,E2 22378.092} C_VEL
LIN {X 0,Y 521.455,Z 1035.359,A -85,B 0,C 180,E1 22376.084,E2 22376.084} C_VEL
LIN {X 0,Y 525.702,Z 1018.413,A -85,B 0,C 180,E1 22374.543,E2 22374.543} C_VEL
LIN {X 0,Y 530.103,Z 1000.137,A -85,B 0,C 180,E1 22373.063,E2 22373.063} C_VEL
LIN {X 0,Y 534.903,Z 979.239,A -85,B 0,C 180,E1 22371.573,E2 22371.573} C_VEL
LIN {X 0,Y 540.286,Z 953.563,A -85,B 0,C 180,E1 22370.012,E2 22370.012} C_VEL
LIN {X 0,Y 544.196,Z 932.933,A -85,B 0,C 180,E1 22368.941,E2 22368.941} C_VEL
LIN {X 0,Y 547.576,Z 913.402,A -85,B 0,C 180,E1 22368.064,E2 22368.064} C_VEL
LIN {X 0,Y 550.747,Z 892.842,A -85,B 0,C 180,E1 22367.272,E2 22367.272} C_VEL
LIN {X 0,Y 553.685,Z 870.826,A -85,B 0,C 180,E1 22366.559,E2 22366.559} C_VEL
LIN {X 0,Y 556.823,Z 841.791,A -85,B 0,C 180,E1 22365.823,E2 22365.823} C_VEL
LIN {X 0,Y 558.693,Z 817.717,A -85,B 0,C 180,E1 22365.375,E2 22365.375} C_VEL
LIN {X 0,Y 566.941,Z 621.303,A -85,B 0,C 180,E1 22362.454,E2 22362.454} C_VEL
LIN {X 0,Y 573.868,Z 458.802,A -85,B 0,C 180,E1 22360.011,E2 22360.011} C_VEL
LIN {X 0,Y 558.484,Z 436.266,A -85,B 0,C 180,E1 22357.195,E2 22357.195} C_VEL
LIN {X 0,Y 547.831,Z 422.233,A -85,B 0,C 180,E1 22355.063,E2 22355.063} C_VEL
LIN {X 0,Y 539.676,Z 411.781,A -85,B 0,C 180,E1 22353.29,E2 22353.29} C_VEL
LIN {X 0,Y 535.332,Z 406.408,A -85,B 0,C 180,E1 22352.289,E2 22352.289} C_VEL
LIN {X 0,Y 531.639,Z 401.78,A -85,B 0,C 180,E1 22351.398,E2 22351.398} C_VEL
LIN {X 0,Y 527.262,Z 396.44,A -85,B 0,C 180,E1 22350.294,E2 22350.294} C_VEL
LIN {X 0,Y 522.863,Z 391.121,A -85,B 0,C 180,E1 22349.123,E2 22349.123} C_VEL
LIN {X 0,Y 519.178,Z 386.813,A -85,B 0,C 180,E1 22348.092,E2 22348.092} C_VEL
LIN {X 0,Y 517.933,Z 385.238,A -85,B 0,C 180,E1 22347.727,E2 22347.727} C_VEL
LIN {X 0,Y 514.408,Z 381.493,A -85,B 0,C 180,E1 22346.68,E2 22346.68} C_VEL
LIN {X 0,Y 512.932,Z 379.311,A -85,B 0,C 180,E1 22346.202,E2 22346.202} C_VEL
LIN {X 0,Y 509.493,Z 376.168,A -85,B 0,C 180,E1 22345.113,E2 22345.113} C_VEL
LIN {X 0,Y 507.611,Z 373.144,A -85,B 0,C 180,E1 22344.435,E2 22344.435} C_VEL
LIN {X 0,Y 504.324,Z 370.591,A -85,B 0,C 180,E1 22343.3,E2 22343.3} C_VEL
LIN {X 0,Y 502.149,Z 366.871,A -85,B 0,C 180,E1 22342.416,E2 22342.416} C_VEL
LIN {X 0,Y 498.34,Z 364.115,A -85,B 0,C 180,E1 22340.925,E2 22340.925} C_VEL
LIN {X 0,Y 496.415,Z 360.999,A -85,B 0,C 180,E1 22340.024,E2 22340.024} C_VEL
LIN {X 0,Y 495.985,Z 359.943,A -85,B 0,C 180,E1 22339.797,E2 22339.797} C_VEL
LIN {X 0,Y 492.41,Z 358.086,A -85,B 0,C 180,E1 22338.162,E2 22338.162} C_VEL
LIN {X 0,Y 490.572,Z 355.395,A -85,B 0,C 180,E1 22337.129,E2 22337.129} C_VEL
LIN {X 0,Y 489.935,Z 353.181,A -85,B 0,C 180,E1 22336.663,E2 22336.663} C_VEL
LIN {X 0,Y 489.933,Z 353.181,A -85,B 0,C 180,E1 22333.334,E2 22333.334} C_VEL
LIN {X 0,Y 489.905,Z 353.184,A -85,B 0,C 180,E1 22329.872,E2 22329.872} C_VEL
LIN {X 0,Y 489.943,Z 353.18,A -85,B 0,C 180,E1 22326.445,E2 22326.445} C_VEL
LIN {X 0,Y 489.936,Z 353.182,A -85,B 0,C 180,E1 22323.042,E2 22323.042} C_VEL
LIN {X 0,Y 489.907,Z 353.188,A -85,B 0,C 180,E1 22319.649,E2 22319.649} C_VEL
LIN {X 0,Y 489.952,Z 353.183,A -85,B 0,C 180,E1 22316.256,E2 22316.256} C_VEL
LIN {X 0,Y 489.934,Z 353.188,A -85,B 0,C 180,E1 22312.849,E2 22312.849} C_VEL
LIN {X 0,Y 490.006,Z 353.447,A -85,B 0,C 180,E1 22310.382,E2 22310.382} C_VEL
LIN {X 0,Y 490.86,Z 356.058,A -85,B 0,C 180,E1 22309.792,E2 22309.792} C_VEL
LIN {X 0,Y 492.996,Z 358.492,A -85,B 0,C 180,E1 22308.654,E2 22308.654} C_VEL
LIN {X 0,Y 496.163,Z 360.19,A -85,B 0,C 180,E1 22307.222,E2 22307.222} C_VEL
LIN {X 0,Y 497.816,Z 363.462,A -85,B 0,C 180,E1 22306.408,E2 22306.408} C_VEL
LIN {X 0,Y 500.5,Z 365.957,A -85,B 0,C 180,E1 22305.302,E2 22305.302} C_VEL
LIN {X 0,Y 502.172,Z 367.019,A -85,B 0,C 180,E1 22304.673,E2 22304.673} C_VEL
LIN {X 0,Y 504.269,Z 370.549,A -85,B 0,C 180,E1 22303.824,E2 22303.824} C_VEL
LIN {X 0,Y 507.541,Z 373.047,A -85,B 0,C 180,E1 22302.694,E2 22302.694} C_VEL
LIN {X 0,Y 510.604,Z 377.428,A -85,B 0,C 180,E1 22301.622,E2 22301.622} C_VEL
LIN {X 0,Y 513.4,Z 379.869,A -85,B 0,C 180,E1 22300.754,E2 22300.754} C_VEL
LIN {X 0,Y 516.5,Z 384.025,A -85,B 0,C 180,E1 22299.784,E2 22299.784} C_VEL
LIN {X 0,Y 518.839,Z 386.298,A -85,B 0,C 180,E1 22299.113,E2 22299.113} C_VEL
LIN {X 0,Y 522.461,Z 390.741,A -85,B 0,C 180,E1 22298.087,E2 22298.087} C_VEL
LIN {X 0,Y 524.252,Z 392.73,A -85,B 0,C 180,E1 22297.606,E2 22297.606} C_VEL
LIN {X 0,Y 529.458,Z 399.035,A -85,B 0,C 180,E1 22296.251,E2 22296.251} C_VEL
LIN {X 0,Y 536.632,Z 408.182,A -85,B 0,C 180,E1 22294.506,E2 22294.506} C_VEL
LIN {X 0,Y 547.77,Z 423.393,A -85,B 0,C 180,E1 22292.022,E2 22292.022} C_VEL
LIN {X 0,Y 559.524,Z 440.32,A -85,B 0,C 180,E1 22289.65,E2 22289.65} C_VEL
LIN {X 0,Y 573.907,Z 461.872,A -85,B 0,C 180,E1 22287.023,E2 22287.023} C_VEL
LIN {X 0,Y 565.692,Z 655.041,A -85,B 0,C 180,E1 22284.129,E2 22284.129} C_VEL
LIN {X 0,Y 558.559,Z 825.678,A -85,B 0,C 180,E1 22281.591,E2 22281.591} C_VEL
LIN {X 0,Y 556.588,Z 850.754,A -85,B 0,C 180,E1 22281.125,E2 22281.125} C_VEL
LIN {X 0,Y 553.468,Z 879.016,A -85,B 0,C 180,E1 22280.407,E2 22280.407} C_VEL
LIN {X 0,Y 550.544,Z 900.74,A -85,B 0,C 180,E1 22279.709,E2 22279.709} C_VEL
LIN {X 0,Y 547.39,Z 921.163,A -85,B 0,C 180,E1 22278.927,E2 22278.927} C_VEL
LIN {X 0,Y 543.923,Z 941.268,A -85,B 0,C 180,E1 22278.028,E2 22278.028} C_VEL
LIN {X 0,Y 539.543,Z 964.346,A -85,B 0,C 180,E1 22276.828,E2 22276.828} C_VEL
LIN {X 0,Y 534.165,Z 989.682,A -85,B 0,C 180,E1 22275.265,E2 22275.265} C_VEL
LIN {X 0,Y 529.659,Z 1009.439,A -85,B 0,C 180,E1 22273.852,E2 22273.852} C_VEL
LIN {X 0,Y 525.365,Z 1027.402,A -85,B 0,C 180,E1 22272.4,E2 22272.4} C_VEL
LIN {X 0,Y 520.849,Z 1045.614,A -85,B 0,C 180,E1 22270.744,E2 22270.744} C_VEL
LIN {X 0,Y 515.22,Z 1067.566,A -85,B 0,C 180,E1 22268.46,E2 22268.46} C_VEL
LIN {X 0,Y 510.713,Z 1084.882,A -85,B 0,C 180,E1 22266.385,E2 22266.385} C_VEL
LIN {X 0,Y 507.007,Z 1099.201,A -85,B 0,C 180,E1 22264.471,E2 22264.471} C_VEL
LIN {X 0,Y 503.534,Z 1112.992,A -85,B 0,C 180,E1 22262.421,E2 22262.421} C_VEL
LIN {X 0,Y 500.152,Z 1126.884,A -85,B 0,C 180,E1 22260.117,E2 22260.117} C_VEL
LIN {X 0,Y 496.351,Z 1143.522,A -85,B 0,C 180,E1 22256.952,E2 22256.952} C_VEL
LIN {X 0,Y 494.007,Z 1154.651,A -85,B 0,C 180,E1 22254.514,E2 22254.514} C_VEL
LIN {X 0,Y 492.162,Z 1164.503,A -85,B 0,C 180,E1 22252.076,E2 22252.076} C_VEL
LIN {X 0,Y 490.734,Z 1173.1,A -85,B 0,C 180,E1 22249.644,E2 22249.644} C_VEL
LIN {X 0,Y 489.581,Z 1181.268,A -85,B 0,C 180,E1 22246.98,E2 22246.98} C_VEL
LIN {X 0,Y 488.655,Z 1189.787,A -85,B 0,C 180,E1 22243.61,E2 22243.61} C_VEL
LIN {X 0,Y 488.216,Z 1195.271,A -85,B 0,C 180,E1 22240.86,E2 22240.86} C_VEL
LIN {X 0,Y 488.027,Z 1199.189,A -85,B 0,C 180,E1 22238.364,E2 22238.364} C_VEL
LIN {X 0,Y 487.942,Z 1202.078,A -85,B 0,C 180,E1 22235.881,E2 22235.881} C_VEL
LIN {X 0,Y 487.915,Z 1203.956,A -85,B 0,C 180,E1 22233.407,E2 22233.407} C_VEL
LIN {X 0,Y 487.906,Z 1204.826,A -85,B 0,C 180,E1 22230.939,E2 22230.939} C_VEL
LIN {X 0,Y 487.909,Z 1204.712,A -85,B 0,C 180,E1 22228.473,E2 22228.473} C_VEL
LIN {X 0,Y 487.919,Z 1203.478,A -85,B 0,C 180,E1 22225.769,E2 22225.769} C_VEL
LIN {X 0,Y 487.99,Z 1200.466,A -85,B 0,C 180,E1 22222.583,E2 22222.583} C_VEL
LIN {X 0,Y 488.162,Z 1196.303,A -85,B 0,C 180,E1 22219.735,E2 22219.735} C_VEL
LIN {X 0,Y 488.48,Z 1191.567,A -85,B 0,C 180,E1 22217.229,E2 22217.229} C_VEL
LIN {X 0,Y 489.055,Z 1185.744,A -85,B 0,C 180,E1 22214.708,E2 22214.708} C_VEL
LIN {X 0,Y 489.941,Z 1178.44,A -85,B 0,C 180,E1 22212.052,E2 22212.052} C_VEL
LIN {X 0,Y 491.556,Z 1168.185,A -85,B 0,C 180,E1 22208.898,E2 22208.898} C_VEL
LIN {X 0,Y 493.578,Z 1156.892,A -85,B 0,C 180,E1 22206.013,E2 22206.013} C_VEL
LIN {X 0,Y 495.704,Z 1146.403,A -85,B 0,C 180,E1 22203.657,E2 22203.657} C_VEL
LIN {X 0,Y 498.391,Z 1134.356,A -85,B 0,C 180,E1 22201.25,E2 22201.25} C_VEL
LIN {X 0,Y 502.03,Z 1119.098,A -85,B 0,C 180,E1 22198.547,E2 22198.547} C_VEL
LIN {X 0,Y 506.371,Z 1101.706,A -85,B 0,C 180,E1 22195.891,E2 22195.891} C_VEL
LIN {X 0,Y 510.259,Z 1086.56,A -85,B 0,C 180,E1 22193.838,E2 22193.838} C_VEL
LIN {X 0,Y 514.303,Z 1070.988,A -85,B 0,C 180,E1 22191.942,E2 22191.942} C_VEL
LIN {X 0,Y 519.21,Z 1052.214,A -85,B 0,C 180,E1 22189.898,E2 22189.898} C_VEL
LIN {X 0,Y 524.998,Z 1029.566,A -85,B 0,C 180,E1 22187.756,E2 22187.756} C_VEL
LIN {X 0,Y 529.785,Z 1010.261,A -85,B 0,C 180,E1 22186.161,E2 22186.161} C_VEL
LIN {X 0,Y 534.361,Z 991.057,A -85,B 0,C 180,E1 22184.758,E2 22184.758} C_VEL
LIN {X 0,Y 539.843,Z 966.836,A -85,B 0,C 180,E1 22183.213,E2 22183.213} C_VEL
LIN {X 0,Y 544.831,Z 942.002,A -85,B 0,C 180,E1 22181.89,E2 22181.89} C_VEL
LIN {X 0,Y 548.65,Z 921.157,A -85,B 0,C 180,E1 22180.941,E2 22180.941} C_VEL
LIN {X 0,Y 552.007,Z 900.756,A -85,B 0,C 180,E1 22180.149,E2 22180.149} C_VEL
LIN {X 0,Y 555.151,Z 878.863,A -85,B 0,C 180,E1 22179.435,E2 22179.435} C_VEL
LIN {X 0,Y 558.479,Z 850.691,A -85,B 0,C 180,E1 22178.712,E2 22178.712} C_VEL
LIN {X 0,Y 560.598,Z 825.627,A -85,B 0,C 180,E1 22178.239,E2 22178.239} C_VEL
LIN {X 0,Y 569.793,Z 632.365,A -85,B 0,C 180,E1 22175.303,E2 22175.303} C_VEL
LIN {X 0,Y 578.257,Z 462.625,A -85,B 0,C 180,E1 22172.708,E2 22172.708} C_VEL
LIN {X 0,Y 570.131,Z 449.709,A -85,B 0,C 180,E1 22170.95,E2 22170.95} C_VEL
LIN {X 0,Y 559.762,Z 434.466,A -85,B 0,C 180,E1 22168.486,E2 22168.486} C_VEL
LIN {X 0,Y 552.336,Z 424.465,A -85,B 0,C 180,E1 22166.532,E2 22166.532} C_VEL
LIN {X 0,Y 547.969,Z 418.565,A -85,B 0,C 180,E1 22165.276,E2 22165.276} C_VEL
LIN {X 0,Y 544.392,Z 413.796,A -85,B 0,C 180,E1 22164.179,E2 22164.179} C_VEL
LIN {X 0,Y 537.873,Z 405.614,A -85,B 0,C 180,E1 22161.999,E2 22161.999} C_VEL
LIN {X 0,Y 534.298,Z 401.563,A -85,B 0,C 180,E1 22160.682,E2 22160.682} C_VEL
LIN {X 0,Y 533.074,Z 399.841,A -85,B 0,C 180,E1 22160.19,E2 22160.19} C_VEL
LIN {X 0,Y 529.748,Z 396.601,A -85,B 0,C 180,E1 22158.83,E2 22158.83} C_VEL
LIN {X 0,Y 527.958,Z 393.737,A -85,B 0,C 180,E1 22157.981,E2 22157.981} C_VEL
LIN {X 0,Y 524.316,Z 390.587,A -85,B 0,C 180,E1 22156.223,E2 22156.223} C_VEL
LIN {X 0,Y 522.415,Z 387.362,A -85,B 0,C 180,E1 22155.088,E2 22155.088} C_VEL
LIN {X 0,Y 519.245,Z 385.144,A -85,B 0,C 180,E1 22153.134,E2 22153.134} C_VEL
LIN {X 0,Y 517.25,Z 381.955,A -85,B 0,C 180,E1 22151.485,E2 22151.485} C_VEL
LIN {X 0,Y 516.829,Z 380.783,A -85,B 0,C 180,E1 22151.042,E2 22151.042} C_VEL
LIN {X 0,Y 512.536,Z 378.096,A -85,B 0,C 180,E1 22144.364,E2 22144.364} C_VEL
LIN {X 0,Y 512.816,Z 378.332,A -85,B 0,C 180,E1 22141.229,E2 22141.229} C_VEL
LIN {X 0,Y 516.96,Z 381.079,A -85,B 0,C 180,E1 22135.618,E2 22135.618} C_VEL
LIN {X 0,Y 518.599,Z 384.425,A -85,B 0,C 180,E1 22134.135,E2 22134.135} C_VEL
LIN {X 0,Y 521.762,Z 387.056,A -85,B 0,C 180,E1 22132.069,E2 22132.069} C_VEL
LIN {X 0,Y 522.711,Z 387.737,A -85,B 0,C 180,E1 22131.53,E2 22131.53} C_VEL
LIN {X 0,Y 525.04,Z 391.452,A -85,B 0,C 180,E1 22130.186,E2 22130.186} C_VEL
LIN {X 0,Y 528.364,Z 394.273,A -85,B 0,C 180,E1 22128.622,E2 22128.622} C_VEL
LIN {X 0,Y 531.219,Z 398.307,A -85,B 0,C 180,E1 22127.333,E2 22127.333} C_VEL
LIN {X 0,Y 533.726,Z 400.616,A -85,B 0,C 180,E1 22126.346,E2 22126.346} C_VEL
LIN {X 0,Y 537.111,Z 404.965,A -85,B 0,C 180,E1 22125.058,E2 22125.058} C_VEL
LIN {X 0,Y 538.939,Z 406.861,A -85,B 0,C 180,E1 22124.422,E2 22124.422} C_VEL
LIN {X 0,Y 542.8,Z 411.477,A -85,B 0,C 180,E1 22123.134,E2 22123.134} C_VEL
LIN {X 0,Y 548.891,Z 419.01,A -85,B 0,C 180,E1 22121.272,E2 22121.272} C_VEL
LIN {X 0,Y 554.129,Z 425.597,A -85,B 0,C 180,E1 22119.812,E2 22119.812} C_VEL
LIN {X 0,Y 561.018,Z 434.412,A -85,B 0,C 180,E1 22118.048,E2 22118.048} C_VEL
LIN {X 0,Y 568.732,Z 444.971,A -85,B 0,C 180,E1 22116.231,E2 22116.231} C_VEL
LIN {X 0,Y 578.245,Z 459.594,A -85,B 0,C 180,E1 22114.163,E2 22114.163} C_VEL
LIN {X 0,Y 567.751,Z 671.179,A -85,B 0,C 180,E1 22110.932,E2 22110.932} C_VEL
LIN {X 0,Y 560.72,Z 818.458,A -85,B 0,C 180,E1 22108.693,E2 22108.693} C_VEL
LIN {X 0,Y 558.55,Z 844.199,A -85,B 0,C 180,E1 22108.201,E2 22108.201} C_VEL
LIN {X 0,Y 555.295,Z 871.662,A -85,B 0,C 180,E1 22107.483,E2 22107.483} C_VEL
LIN {X 0,Y 552.349,Z 892.373,A -85,B 0,C 180,E1 22106.804,E2 22106.804} C_VEL
LIN {X 0,Y 548.995,Z 912.918,A -85,B 0,C 180,E1 22106.003,E2 22106.003} C_VEL
LIN {X 0,Y 545.397,Z 932.58,A -85,B 0,C 180,E1 22105.11,E2 22105.11} C_VEL
LIN {X 0,Y 541.226,Z 953.423,A -85,B 0,C 180,E1 22104.014,E2 22104.014} C_VEL
LIN {X 0,Y 535.755,Z 978.364,A -85,B 0,C 180,E1 22102.482,E2 22102.482} C_VEL
LIN {X 0,Y 530.594,Z 999.869,A -85,B 0,C 180,E1 22100.93,E2 22100.93} C_VEL
LIN {X 0,Y 525.972,Z 1018.356,A -85,B 0,C 180,E1 22099.415,E2 22099.415} C_VEL
LIN {X 0,Y 521.341,Z 1036.339,A -85,B 0,C 180,E1 22097.756,E2 22097.756} C_VEL
LIN {X 0,Y 515.719,Z 1057.723,A -85,B 0,C 180,E1 22095.517,E2 22095.517} C_VEL
LIN {X 0,Y 513.757,Z 1065.05,A -85,B 0,C 180,E1 22094.659,E2 22094.659} C_VEL
LIN {X 0,Y 511.516,Z 1070.525,A -85,B 0,C 180,E1 22094.086,E2 22094.086} C_VEL
LIN {X 0,Y 502.353,Z 1084.917,A -85,B 0,C 180,E1 22092.656,E2 22092.656} C_VEL
LIN {X 0,Y 500.544,Z 1089.089,A -85,B 0,C 180,E1 22092.108,E2 22092.108} C_VEL
LIN {X 0,Y 496.624,Z 1103.664,A -85,B 0,C 180,E1 22089.906,E2 22089.906} C_VEL
LIN {X 0,Y 492.627,Z 1119.052,A -85,B 0,C 180,E1 22087.283,E2 22087.283} C_VEL
LIN {X 0,Y 488.821,Z 1134.541,A -85,B 0,C 180,E1 22084.229,E2 22084.229} C_VEL
LIN {X 0,Y 485.899,Z 1147.573,A -85,B 0,C 180,E1 22081.235,E2 22081.235} C_VEL
LIN {X 0,Y 483.871,Z 1157.839,A -85,B 0,C 180,E1 22078.511,E2 22078.511} C_VEL
LIN {X 0,Y 482.127,Z 1168.291,A -85,B 0,C 180,E1 22075.28,E2 22075.28} C_VEL
LIN {X 0,Y 481.094,Z 1176.136,A -85,B 0,C 180,E1 22072.35,E2 22072.35} C_VEL
LIN {X 0,Y 480.502,Z 1181.802,A -85,B 0,C 180,E1 22069.827,E2 22069.827} C_VEL
LIN {X 0,Y 480.167,Z 1186.617,A -85,B 0,C 180,E1 22067.199,E2 22067.199} C_VEL
LIN {X 0,Y 479.991,Z 1190.626,A -85,B 0,C 180,E1 22064.352,E2 22064.352} C_VEL
LIN {X 0,Y 479.917,Z 1193.583,A -85,B 0,C 180,E1 22061.092,E2 22061.092} C_VEL
LIN {X 0,Y 479.913,Z 1194.742,A -85,B 0,C 180,E1 22058.386,E2 22058.386} C_VEL
LIN {X 0,Y 479.913,Z 1194.826,A -85,B 0,C 180,E1 22055.979,E2 22055.979} C_VEL
LIN {X 0,Y 479.912,Z 1193.942,A -85,B 0,C 180,E1 22053.464,E2 22053.464} C_VEL
LIN {X 0,Y 479.944,Z 1192.062,A -85,B 0,C 180,E1 22050.955,E2 22050.955} C_VEL
LIN {X 0,Y 480.044,Z 1189.044,A -85,B 0,C 180,E1 22048.329,E2 22048.329} C_VEL
LIN {X 0,Y 480.359,Z 1183.877,A -85,B 0,C 180,E1 22045.104,E2 22045.104} C_VEL
LIN {X 0,Y 480.899,Z 1177.758,A -85,B 0,C 180,E1 22042.233,E2 22042.233} C_VEL
LIN {X 0,Y 481.73,Z 1170.989,A -85,B 0,C 180,E1 22039.597,E2 22039.597} C_VEL
LIN {X 0,Y 483.008,Z 1162.702,A -85,B 0,C 180,E1 22036.838,E2 22036.838} C_VEL
LIN {X 0,Y 485.238,Z 1150.771,A -85,B 0,C 180,E1 22033.48,E2 22033.48} C_VEL
LIN {X 0,Y 487.941,Z 1138.217,A -85,B 0,C 180,E1 22030.488,E2 22030.488} C_VEL
LIN {X 0,Y 491.447,Z 1123.57,A -85,B 0,C 180,E1 22027.474,E2 22027.474} C_VEL
LIN {X 0,Y 495.91,Z 1106.37,A -85,B 0,C 180,E1 22024.439,E2 22024.439} C_VEL
LIN {X 0,Y 500.195,Z 1090.311,A -85,B 0,C 180,E1 22021.982,E2 22021.982} C_VEL
LIN {X 0,Y 504.405,Z 1074.99,A -85,B 0,C 180,E1 22019.9,E2 22019.9} C_VEL
LIN {X 0,Y 509.941,Z 1054.961,A -85,B 0,C 180,E1 22017.504,E2 22017.504} C_VEL
LIN {X 0,Y 514.997,Z 1035.978,A -85,B 0,C 180,E1 22015.543,E2 22015.543} C_VEL
LIN {X 0,Y 519.584,Z 1018.297,A -85,B 0,C 180,E1 22013.925,E2 22013.925} C_VEL
LIN {X 0,Y 524.291,Z 999.402,A -85,B 0,C 180,E1 22012.392,E2 22012.392} C_VEL
LIN {X 0,Y 529.885,Z 975.827,A -85,B 0,C 180,E1 22010.723,E2 22010.723} C_VEL
LIN {X 0,Y 534.783,Z 952.71,A -85,B 0,C 180,E1 22009.34,E2 22009.34} C_VEL
LIN {X 0,Y 538.721,Z 932.47,A -85,B 0,C 180,E1 22008.289,E2 22008.289} C_VEL
LIN {X 0,Y 542.208,Z 912.833,A -85,B 0,C 180,E1 22007.409,E2 22007.409} C_VEL
LIN {X 0,Y 545.486,Z 892.146,A -85,B 0,C 180,E1 22006.615,E2 22006.615} C_VEL
LIN {X 0,Y 548.705,Z 868.571,A -85,B 0,C 180,E1 22005.859,E2 22005.859} C_VEL
LIN {X 0,Y 551.754,Z 840.24,A -85,B 0,C 180,E1 22005.158,E2 22005.158} C_VEL
LIN {X 0,Y 553.576,Z 817.059,A -85,B 0,C 180,E1 22004.731,E2 22004.731} C_VEL
LIN {X 0,Y 562.186,Z 618.922,A -85,B 0,C 180,E1 22001.769,E2 22001.769} C_VEL
LIN {X 0,Y 569.143,Z 463.169,A -85,B 0,C 180,E1 21999.427,E2 21999.427} C_VEL
LIN {X 0,Y 554.401,Z 441.418,A -85,B 0,C 180,E1 21996.654,E2 21996.654} C_VEL
LIN {X 0,Y 542.115,Z 425.138,A -85,B 0,C 180,E1 21994.105,E2 21994.105} C_VEL
LIN {X 0,Y 533.463,Z 414.191,A -85,B 0,C 180,E1 21992.13,E2 21992.13} C_VEL
LIN {X 0,Y 528.784,Z 408.384,A -85,B 0,C 180,E1 21990.985,E2 21990.985} C_VEL
LIN {X 0,Y 524.862,Z 403.522,A -85,B 0,C 180,E1 21989.974,E2 21989.974} C_VEL
LIN {X 0,Y 520.61,Z 398.342,A -85,B 0,C 180,E1 21988.821,E2 21988.821} C_VEL
LIN {X 0,Y 516.72,Z 393.583,A -85,B 0,C 180,E1 21987.704,E2 21987.704} C_VEL
LIN {X 0,Y 512.115,Z 388.414,A -85,B 0,C 180,E1 21986.309,E2 21986.309} C_VEL
LIN {X 0,Y 510.801,Z 386.677,A -85,B 0,C 180,E1 21985.882,E2 21985.882} C_VEL
LIN {X 0,Y 507.36,Z 383.237,A -85,B 0,C 180,E1 21984.758,E2 21984.758} C_VEL
LIN {X 0,Y 505.719,Z 380.699,A -85,B 0,C 180,E1 21984.159,E2 21984.159} C_VEL
LIN {X 0,Y 502.356,Z 377.802,A -85,B 0,C 180,E1 21982.962,E2 21982.962} C_VEL
LIN {X 0,Y 500.201,Z 374.277,A -85,B 0,C 180,E1 21982.074,E2 21982.074} C_VEL
LIN {X 0,Y 496.868,Z 371.824,A -85,B 0,C 180,E1 21980.743,E2 21980.743} C_VEL
LIN {X 0,Y 494.726,Z 368.437,A -85,B 0,C 180,E1 21979.726,E2 21979.726} C_VEL
LIN {X 0,Y 494.239,Z 367.678,A -85,B 0,C 180,E1 21979.485,E2 21979.485} C_VEL
LIN {X 0,Y 490.795,Z 365.576,A -85,B 0,C 180,E1 21977.855,E2 21977.855} C_VEL
LIN {X 0,Y 488.931,Z 362.565,A -85,B 0,C 180,E1 21976.759,E2 21976.759} C_VEL
LIN {X 0,Y 488.34,Z 361.029,A -85,B 0,C 180,E1 21976.352,E2 21976.352} C_VEL
LIN {X 0,Y 484.674,Z 359.245,A -85,B 0,C 180,E1 21974.09,E2 21974.09} C_VEL
LIN {X 0,Y 482.383,Z 355.906,A -85,B 0,C 180,E1 21972.145,E2 21972.145} C_VEL
LIN {X 0,Y 481.974,Z 354.196,A -85,B 0,C 180,E1 21971.609,E2 21971.609} C_VEL
LIN {X 0,Y 481.972,Z 354.197,A -85,B 0,C 180,E1 21967.99,E2 21967.99} C_VEL
LIN {X 0,Y 482.027,Z 354.186,A -85,B 0,C 180,E1 21964.64,E2 21964.64} C_VEL
LIN {X 0,Y 481.993,Z 354.19,A -85,B 0,C 180,E1 21961.07,E2 21961.07} C_VEL
LIN {X 0,Y 481.973,Z 354.189,A -85,B 0,C 180,E1 21957.622,E2 21957.622} C_VEL
LIN {X 0,Y 481.989,Z 354.312,A -85,B 0,C 180,E1 21955.449,E2 21955.449} C_VEL
LIN {X 0,Y 482.817,Z 356.774,A -85,B 0,C 180,E1 21954.533,E2 21954.533} C_VEL
LIN {X 0,Y 484.847,Z 359.367,A -85,B 0,C 180,E1 21952.892,E2 21952.892} C_VEL
LIN {X 0,Y 488.52,Z 361.356,A -85,B 0,C 180,E1 21950.635,E2 21950.635} C_VEL
LIN {X 0,Y 489.85,Z 364.384,A -85,B 0,C 180,E1 21949.771,E2 21949.771} C_VEL
LIN {X 0,Y 492.741,Z 366.963,A -85,B 0,C 180,E1 21948.292,E2 21948.292} C_VEL
LIN {X 0,Y 494.603,Z 368.049,A -85,B 0,C 180,E1 21947.448,E2 21947.448} C_VEL
LIN {X 0,Y 496.818,Z 371.795,A -85,B 0,C 180,E1 21946.38,E2 21946.38} C_VEL
LIN {X 0,Y 500.129,Z 374.277,A -85,B 0,C 180,E1 21945.054,E2 21945.054} C_VEL
LIN {X 0,Y 502.991,Z 378.556,A -85,B 0,C 180,E1 21943.9,E2 21943.9} C_VEL
LIN {X 0,Y 506.071,Z 381.104,A -85,B 0,C 180,E1 21942.82,E2 21942.82} C_VEL
LIN {X 0,Y 508.975,Z 385.115,A -85,B 0,C 180,E1 21941.799,E2 21941.799} C_VEL
LIN {X 0,Y 511.482,Z 387.41,A -85,B 0,C 180,E1 21941.005,E2 21941.005} C_VEL
LIN {X 0,Y 514.823,Z 391.723,A -85,B 0,C 180,E1 21939.952,E2 21939.952} C_VEL
LIN {X 0,Y 516.777,Z 393.697,A -85,B 0,C 180,E1 21939.381,E2 21939.381} C_VEL
LIN {X 0,Y 520.551,Z 398.268,A -85,B 0,C 180,E1 21938.299,E2 21938.299} C_VEL
LIN {X 0,Y 522.587,Z 400.769,A -85,B 0,C 180,E1 21937.738,E2 21937.738} C_VEL
LIN {X 0,Y 527.091,Z 406.156,A -85,B 0,C 180,E1 21936.553,E2 21936.553} C_VEL
LIN {X 0,Y 534.284,Z 415.462,A -85,B 0,C 180,E1 21934.772,E2 21934.772} C_VEL
LIN {X 0,Y 545.098,Z 430.416,A -85,B 0,C 180,E1 21932.319,E2 21932.319} C_VEL
LIN {X 0,Y 556.507,Z 447.049,A -85,B 0,C 180,E1 21929.974,E2 21929.974} C_VEL
LIN {X 0,Y 569.151,Z 466.173,A -85,B 0,C 180,E1 21927.611,E2 21927.611} C_VEL
LIN {X 0,Y 559.762,Z 678.621,A -85,B 0,C 180,E1 21924.424,E2 21924.424} C_VEL
LIN {X 0,Y 553.38,Z 825.765,A -85,B 0,C 180,E1 21922.222,E2 21922.222} C_VEL
LIN {X 0,Y 551.277,Z 851.72,A -85,B 0,C 180,E1 21921.736,E2 21921.736} C_VEL
LIN {X 0,Y 548.106,Z 879.326,A -85,B 0,C 180,E1 21921.028,E2 21921.028} C_VEL
LIN {X 0,Y 545.12,Z 900.866,A -85,B 0,C 180,E1 21920.333,E2 21920.333} C_VEL
LIN {X 0,Y 541.801,Z 921.672,A -85,B 0,C 180,E1 21919.533,E2 21919.533} C_VEL
LIN {X 0,Y 538.03,Z 942.814,A -85,B 0,C 180,E1 21918.578,E2 21918.578} C_VEL
LIN {X 0,Y 532.866,Z 968.776,A -85,B 0,C 180,E1 21917.194,E2 21917.194} C_VEL
LIN {X 0,Y 527.968,Z 990.841,A -85,B 0,C 180,E1 21915.798,E2 21915.798} C_VEL
LIN {X 0,Y 523.679,Z 1009.081,A -85,B 0,C 180,E1 21914.484,E2 21914.484} C_VEL
LIN {X 0,Y 519.29,Z 1026.84,A -85,B 0,C 180,E1 21913.044,E2 21913.044} C_VEL
LIN {X 0,Y 514.727,Z 1044.625,A -85,B 0,C 180,E1 21911.424,E2 21911.424} C_VEL
LIN {X 0,Y 509.269,Z 1065.315,A -85,B 0,C 180,E1 21909.292,E2 21909.292} C_VEL
LIN {X 0,Y 504.067,Z 1084.365,A -85,B 0,C 180,E1 21907.006,E2 21907.006} C_VEL
LIN {X 0,Y 500.079,Z 1099.098,A -85,B 0,C 180,E1 21905.017,E2 21905.017} C_VEL
LIN {X 0,Y 496.431,Z 1112.892,A -85,B 0,C 180,E1 21902.943,E2 21902.943} C_VEL
LIN {X 0,Y 492.892,Z 1126.786,A -85,B 0,C 180,E1 21900.608,E2 21900.608} C_VEL
LIN {X 0,Y 488.867,Z 1143.426,A -85,B 0,C 180,E1 21897.399,E2 21897.399} C_VEL
LIN {X 0,Y 486.292,Z 1155.074,A -85,B 0,C 180,E1 21894.799,E2 21894.799} C_VEL
LIN {X 0,Y 484.363,Z 1164.872,A -85,B 0,C 180,E1 21892.323,E2 21892.323} C_VEL
LIN {X 0,Y 482.804,Z 1173.883,A -85,B 0,C 180,E1 21889.728,E2 21889.728} C_VEL
LIN {X 0,Y 481.434,Z 1183.318,A -85,B 0,C 180,E1 21886.53,E2 21886.53} C_VEL
LIN {X 0,Y 480.634,Z 1190.547,A -85,B 0,C 180,E1 21883.473,E2 21883.473} C_VEL
LIN {X 0,Y 480.227,Z 1195.474,A -85,B 0,C 180,E1 21880.922,E2 21880.922} C_VEL
LIN {X 0,Y 480.03,Z 1199.346,A -85,B 0,C 180,E1 21878.384,E2 21878.384} C_VEL
LIN {X 0,Y 479.942,Z 1202.188,A -85,B 0,C 180,E1 21875.859,E2 21875.859} C_VEL
LIN {X 0,Y 479.915,Z 1204.021,A -85,B 0,C 180,E1 21873.344,E2 21873.344} C_VEL
LIN {X 0,Y 479.898,Z 1204.871,A -85,B 0,C 180,E1 21870.716,E2 21870.716} C_VEL
LIN {X 0,Y 479.909,Z 1204.548,A -85,B 0,C 180,E1 21867.612,E2 21867.612} C_VEL
LIN {X 0,Y 479.935,Z 1202.528,A -85,B 0,C 180,E1 21864.501,E2 21864.501} C_VEL
LIN {X 0,Y 480.019,Z 1199.664,A -85,B 0,C 180,E1 21861.857,E2 21861.857} C_VEL
LIN {X 0,Y 480.205,Z 1195.887,A -85,B 0,C 180,E1 21859.321,E2 21859.321} C_VEL
LIN {X 0,Y 480.582,Z 1191.055,A -85,B 0,C 180,E1 21856.77,E2 21856.77} C_VEL
LIN {X 0,Y 481.216,Z 1185.033,A -85,B 0,C 180,E1 21854.164,E2 21854.164} C_VEL
LIN {X 0,Y 482.446,Z 1176.311,A -85,B 0,C 180,E1 21851.012,E2 21851.012} C_VEL
LIN {X 0,Y 484.187,Z 1165.794,A -85,B 0,C 180,E1 21847.924,E2 21847.924} C_VEL
LIN {X 0,Y 486.132,Z 1155.839,A -85,B 0,C 180,E1 21845.384,E2 21845.384} C_VEL
LIN {X 0,Y 488.471,Z 1145.144,A -85,B 0,C 180,E1 21842.973,E2 21842.973} C_VEL
LIN {X 0,Y 491.522,Z 1132.171,A -85,B 0,C 180,E1 21840.376,E2 21840.376} C_VEL
LIN {X 0,Y 495.847,Z 1115.173,A -85,B 0,C 180,E1 21837.426,E2 21837.426} C_VEL
LIN {X 0,Y 499.625,Z 1100.741,A -85,B 0,C 180,E1 21835.226,E2 21835.226} C_VEL
LIN {X 0,Y 503.811,Z 1085.247,A -85,B 0,C 180,E1 21833.113,E2 21833.113} C_VEL
LIN {X 0,Y 508.538,Z 1068.021,A -85,B 0,C 180,E1 21831.012,E2 21831.012} C_VEL
LIN {X 0,Y 514.608,Z 1045.838,A -85,B 0,C 180,E1 21828.654,E2 21828.654} C_VEL
LIN {X 0,Y 519.381,Z 1027.904,A -85,B 0,C 180,E1 21826.986,E2 21826.986} C_VEL
LIN {X 0,Y 524.073,Z 1009.736,A -85,B 0,C 180,E1 21825.482,E2 21825.482} C_VEL
LIN {X 0,Y 528.832,Z 990.521,A -85,B 0,C 180,E1 21824.072,E2 21824.072} C_VEL
LIN {X 0,Y 534.528,Z 966.255,A -85,B 0,C 180,E1 21822.524,E2 21822.524} C_VEL
LIN {X 0,Y 539.636,Z 941.7,A -85,B 0,C 180,E1 21821.214,E2 21821.214} C_VEL
LIN {X 0,Y 543.424,Z 921.741,A -85,B 0,C 180,E1 21820.302,E2 21820.302} C_VEL
LIN {X 0,Y 546.889,Z 901.454,A -85,B 0,C 180,E1 21819.509,E2 21819.509} C_VEL
LIN {X 0,Y 550.065,Z 880.2,A -85,B 0,C 180,E1 21818.81,E2 21818.81} C_VEL
LIN {X 0,Y 553.36,Z 854.125,A -85,B 0,C 180,E1 21818.119,E2 21818.119} C_VEL
LIN {X 0,Y 555.817,Z 826.65,A -85,B 0,C 180,E1 21817.589,E2 21817.589} C_VEL
LIN {X 0,Y 560.667,Z 729.243,A -85,B 0,C 180,E1 21816.095,E2 21816.095} C_VEL
LIN {X 0,Y 571.631,Z 511.669,A -85,B 0,C 180,E1 21812.771,E2 21812.771} C_VEL
LIN {X 0,Y 573.932,Z 466.869,A -85,B 0,C 180,E1 21812.068,E2 21812.068} C_VEL
LIN {X 0,Y 566.383,Z 455.013,A -85,B 0,C 180,E1 21810.384,E2 21810.384} C_VEL
LIN {X 0,Y 557.277,Z 441.369,A -85,B 0,C 180,E1 21808.157,E2 21808.157} C_VEL
LIN {X 0,Y 549.966,Z 431.394,A -85,B 0,C 180,E1 21806.19,E2 21806.19} C_VEL
LIN {X 0,Y 545.584,Z 425.389,A -85,B 0,C 180,E1 21804.899,E2 21804.899} C_VEL
LIN {X 0,Y 542.003,Z 420.579,A -85,B 0,C 180,E1 21803.772,E2 21803.772} C_VEL
LIN {X 0,Y 536.114,Z 413.126,A -85,B 0,C 180,E1 21801.756,E2 21801.756} C_VEL
LIN {X 0,Y 532.481,Z 408.849,A -85,B 0,C 180,E1 21800.385,E2 21800.385} C_VEL
LIN {X 0,Y 531.319,Z 407.367,A -85,B 0,C 180,E1 21799.915,E2 21799.915} C_VEL
LIN {X 0,Y 527.96,Z 403.824,A -85,B 0,C 180,E1 21798.495,E2 21798.495} C_VEL
LIN {X 0,Y 526.536,Z 401.486,A -85,B 0,C 180,E1 21797.803,E2 21797.803} C_VEL
LIN {X 0,Y 522.857,Z 398.156,A -85,B 0,C 180,E1 21795.985,E2 21795.985} C_VEL
LIN {X 0,Y 521.072,Z 395.179,A -85,B 0,C 180,E1 21794.9,E2 21794.9} C_VEL
LIN {X 0,Y 517.77,Z 392.644,A -85,B 0,C 180,E1 21792.788,E2 21792.788} C_VEL
LIN {X 0,Y 515.929,Z 389.368,A -85,B 0,C 180,E1 21791.175,E2 21791.175} C_VEL
LIN {X 0,Y 515.605,Z 388.67,A -85,B 0,C 180,E1 21790.842,E2 21790.842} C_VEL
LIN {X 0,Y 511.559,Z 386.038,A -85,B 0,C 180,E1 21784.372,E2 21784.372} C_VEL
LIN {X 0,Y 511.836,Z 386.28,A -85,B 0,C 180,E1 21781.231,E2 21781.231} C_VEL
LIN {X 0,Y 515.789,Z 388.925,A -85,B 0,C 180,E1 21775.775,E2 21775.775} C_VEL
LIN {X 0,Y 517.469,Z 392.303,A -85,B 0,C 180,E1 21774.233,E2 21774.233} C_VEL
LIN {X 0,Y 520.6,Z 394.933,A -85,B 0,C 180,E1 21772.162,E2 21772.162} C_VEL
LIN {X 0,Y 521.432,Z 395.639,A -85,B 0,C 180,E1 21771.676,E2 21771.676} C_VEL
LIN {X 0,Y 523.95,Z 399.46,A -85,B 0,C 180,E1 21770.221,E2 21770.221} C_VEL
LIN {X 0,Y 526.855,Z 401.912,A -85,B 0,C 180,E1 21768.838,E2 21768.838} C_VEL
LIN {X 0,Y 529.856,Z 406.103,A -85,B 0,C 180,E1 21767.466,E2 21767.466} C_VEL
LIN {X 0,Y 532.134,Z 408.271,A -85,B 0,C 180,E1 21766.554,E2 21766.554} C_VEL
LIN {X 0,Y 535.553,Z 412.635,A -85,B 0,C 180,E1 21765.235,E2 21765.235} C_VEL
LIN {X 0,Y 537.211,Z 414.418,A -85,B 0,C 180,E1 21764.647,E2 21764.647} C_VEL
LIN {X 0,Y 541.184,Z 419.148,A -85,B 0,C 180,E1 21763.303,E2 21763.303} C_VEL
LIN {X 0,Y 547.122,Z 426.704,A -85,B 0,C 180,E1 21761.458,E2 21761.458} C_VEL
LIN {X 0,Y 552.404,Z 433.393,A -85,B 0,C 180,E1 21759.967,E2 21759.967} C_VEL
LIN {X 0,Y 559.609,Z 442.87,A -85,B 0,C 180,E1 21758.1,E2 21758.1} C_VEL
LIN {X 0,Y 566.379,Z 452.272,A -85,B 0,C 180,E1 21756.485,E2 21756.485} C_VEL
LIN {X 0,Y 573.986,Z 464.269,A -85,B 0,C 180,E1 21754.782,E2 21754.782} C_VEL
LIN {X 0,Y 562.992,Z 677.983,A -85,B 0,C 180,E1 21751.508,E2 21751.508} C_VEL
LIN {X 0,Y 556,Z 818.831,A -85,B 0,C 180,E1 21749.356,E2 21749.356} C_VEL
LIN {X 0,Y 553.654,Z 845.753,A -85,B 0,C 180,E1 21748.837,E2 21748.837} C_VEL
LIN {X 0,Y 550.316,Z 872.511,A -85,B 0,C 180,E1 21748.127,E2 21748.127} C_VEL
LIN {X 0,Y 547.219,Z 893.442,A -85,B 0,C 180,E1 21747.434,E2 21747.434} C_VEL
LIN {X 0,Y 543.834,Z 913.426,A -85,B 0,C 180,E1 21746.651,E2 21746.651} C_VEL
LIN {X 0,Y 540.096,Z 933.147,A -85,B 0,C 180,E1 21745.75,E2 21745.75} C_VEL
LIN {X 0,Y 535.529,Z 955.111,A -85,B 0,C 180,E1 21744.584,E2 21744.584} C_VEL
LIN {X 0,Y 529.552,Z 980.936,A -85,B 0,C 180,E1 21742.963,E2 21742.963} C_VEL
LIN {X 0,Y 524.737,Z 1000.278,A -85,B 0,C 180,E1 21741.549,E2 21741.549} C_VEL
LIN {X 0,Y 519.98,Z 1018.541,A -85,B 0,C 180,E1 21740.039,E2 21740.039} C_VEL
LIN {X 0,Y 515.118,Z 1036.615,A -85,B 0,C 180,E1 21738.356,E2 21738.356} C_VEL
LIN {X 0,Y 509.238,Z 1057.904,A -85,B 0,C 180,E1 21736.102,E2 21736.102} C_VEL
LIN {X 0,Y 504.149,Z 1076.062,A -85,B 0,C 180,E1 21733.88,E2 21733.88} C_VEL
LIN {X 0,Y 500.544,Z 1089.089,A -85,B 0,C 180,E1 21732.108,E2 21732.108} C_VEL
LIN {X 0,Y 498.366,Z 1094.041,A -85,B 0,C 180,E1 21731.463,E2 21731.463} C_VEL
LIN {X 0,Y 489.364,Z 1107.193,A -85,B 0,C 180,E1 21729.839,E2 21729.839} C_VEL
LIN {X 0,Y 487.599,Z 1111.019,A -85,B 0,C 180,E1 21729.234,E2 21729.234} C_VEL
LIN {X 0,Y 483.56,Z 1126.041,A -85,B 0,C 180,E1 21726.451,E2 21726.451} C_VEL
LIN {X 0,Y 480.235,Z 1139.382,A -85,B 0,C 180,E1 21723.629,E2 21723.629} C_VEL
LIN {X 0,Y 477.218,Z 1152.821,A -85,B 0,C 180,E1 21720.317,E2 21720.317} C_VEL
LIN {X 0,Y 475.181,Z 1163.152,A -85,B 0,C 180,E1 21717.304,E2 21717.304} C_VEL
LIN {X 0,Y 473.857,Z 1171.185,A -85,B 0,C 180,E1 21714.562,E2 21714.562} C_VEL
LIN {X 0,Y 472.901,Z 1178.568,A -85,B 0,C 180,E1 21711.585,E2 21711.585} C_VEL
LIN {X 0,Y 472.28,Z 1185.171,A -85,B 0,C 180,E1 21708.26,E2 21708.26} C_VEL
LIN {X 0,Y 472.039,Z 1189.376,A -85,B 0,C 180,E1 21705.463,E2 21705.463} C_VEL
LIN {X 0,Y 471.942,Z 1192.162,A -85,B 0,C 180,E1 21702.943,E2 21702.943} C_VEL
LIN {X 0,Y 471.917,Z 1194.009,A -85,B 0,C 180,E1 21700.375,E2 21700.375} C_VEL
LIN {X 0,Y 471.894,Z 1194.854,A -85,B 0,C 180,E1 21697.794,E2 21697.794} C_VEL
LIN {X 0,Y 471.912,Z 1194.648,A -85,B 0,C 180,E1 21694.983,E2 21694.983} C_VEL
LIN {X 0,Y 471.927,Z 1192.937,A -85,B 0,C 180,E1 21691.821,E2 21691.821} C_VEL
LIN {X 0,Y 472.009,Z 1190.114,A -85,B 0,C 180,E1 21689.029,E2 21689.029} C_VEL
LIN {X 0,Y 472.188,Z 1186.522,A -85,B 0,C 180,E1 21686.479,E2 21686.479} C_VEL
LIN {X 0,Y 472.545,Z 1181.928,A -85,B 0,C 180,E1 21683.927,E2 21683.927} C_VEL
LIN {X 0,Y 473.19,Z 1176.044,A -85,B 0,C 180,E1 21681.249,E2 21681.249} C_VEL
LIN {X 0,Y 474.487,Z 1167.346,A -85,B 0,C 180,E1 21677.959,E2 21677.959} C_VEL
LIN {X 0,Y 476.312,Z 1157.074,A -85,B 0,C 180,E1 21674.788,E2 21674.788} C_VEL
LIN {X 0,Y 478.662,Z 1146.053,A -85,B 0,C 180,E1 21671.866,E2 21671.866} C_VEL
LIN {X 0,Y 482.122,Z 1131.642,A -85,B 0,C 180,E1 21668.592,E2 21668.592} C_VEL
LIN {X 0,Y 486.003,Z 1116.752,A -85,B 0,C 180,E1 21665.703,E2 21665.703} C_VEL
LIN {X 0,Y 489.833,Z 1102.755,A -85,B 0,C 180,E1 21663.316,E2 21663.316} C_VEL
LIN {X 0,Y 494.052,Z 1087.952,A -85,B 0,C 180,E1 21661.074,E2 21661.074} C_VEL
LIN {X 0,Y 499.673,Z 1068.395,A -85,B 0,C 180,E1 21658.481,E2 21658.481} C_VEL
LIN {X 0,Y 504.665,Z 1050.655,A -85,B 0,C 180,E1 21656.443,E2 21656.443} C_VEL
LIN {X 0,Y 509.26,Z 1034.022,A -85,B 0,C 180,E1 21654.745,E2 21654.745} C_VEL
LIN {X 0,Y 513.693,Z 1017.489,A -85,B 0,C 180,E1 21653.236,E2 21653.236} C_VEL
LIN {X 0,Y 518.404,Z 999.176,A -85,B 0,C 180,E1 21651.748,E2 21651.748} C_VEL
LIN {X 0,Y 524.182,Z 975.5,A -85,B 0,C 180,E1 21650.07,E2 21650.07} C_VEL
LIN {X 0,Y 529.05,Z 953.259,A -85,B 0,C 180,E1 21648.732,E2 21648.732} C_VEL
LIN {X 0,Y 533.106,Z 933.052,A -85,B 0,C 180,E1 21647.677,E2 21647.677} C_VEL
LIN {X 0,Y 536.696,Z 913.449,A -85,B 0,C 180,E1 21646.792,E2 21646.792} C_VEL
LIN {X 0,Y 540.07,Z 892.811,A -85,B 0,C 180,E1 21645.995,E2 21645.995} C_VEL
LIN {X 0,Y 543.234,Z 870.367,A -85,B 0,C 180,E1 21645.268,E2 21645.268} C_VEL
LIN {X 0,Y 546.523,Z 841.315,A -85,B 0,C 180,E1 21644.536,E2 21644.536} C_VEL
LIN {X 0,Y 548.452,Z 817.581,A -85,B 0,C 180,E1 21644.094,E2 21644.094} C_VEL
LIN {X 0,Y 557.361,Z 619.659,A -85,B 0,C 180,E1 21641.12,E2 21641.12} C_VEL
LIN {X 0,Y 564.336,Z 467.47,A -85,B 0,C 180,E1 21638.813,E2 21638.813} C_VEL
LIN {X 0,Y 551.472,Z 448.186,A -85,B 0,C 180,E1 21636.331,E2 21636.331} C_VEL
LIN {X 0,Y 539.426,Z 432.049,A -85,B 0,C 180,E1 21633.786,E2 21633.786} C_VEL
LIN {X 0,Y 530.771,Z 420.992,A -85,B 0,C 180,E1 21631.772,E2 21631.772} C_VEL
LIN {X 0,Y 526.253,Z 415.319,A -85,B 0,C 180,E1 21630.643,E2 21630.643} C_VEL
LIN {X 0,Y 522.382,Z 410.492,A -85,B 0,C 180,E1 21629.625,E2 21629.625} C_VEL
LIN {X 0,Y 518.374,Z 405.553,A -85,B 0,C 180,E1 21628.516,E2 21628.516} C_VEL
LIN {X 0,Y 514.438,Z 400.598,A -85,B 0,C 180,E1 21627.36,E2 21627.36} C_VEL
LIN {X 0,Y 510.161,Z 395.825,A -85,B 0,C 180,E1 21626.042,E2 21626.042} C_VEL
LIN {X 0,Y 508.859,Z 394.134,A -85,B 0,C 180,E1 21625.613,E2 21625.613} C_VEL
LIN {X 0,Y 505.248,Z 390.298,A -85,B 0,C 180,E1 21624.401,E2 21624.401} C_VEL
LIN {X 0,Y 503.843,Z 388.225,A -85,B 0,C 180,E1 21623.881,E2 21623.881} C_VEL
LIN {X 0,Y 500.403,Z 385.003,A -85,B 0,C 180,E1 21622.622,E2 21622.622} C_VEL
LIN {X 0,Y 498.401,Z 381.886,A -85,B 0,C 180,E1 21621.786,E2 21621.786} C_VEL
LIN {X 0,Y 495.149,Z 379.242,A -85,B 0,C 180,E1 21620.448,E2 21620.448} C_VEL
LIN {X 0,Y 492.826,Z 375.486,A -85,B 0,C 180,E1 21619.312,E2 21619.312} C_VEL
LIN {X 0,Y 489.408,Z 373.28,A -85,B 0,C 180,E1 21617.662,E2 21617.662} C_VEL
LIN {X 0,Y 487.436,Z 370.058,A -85,B 0,C 180,E1 21616.475,E2 21616.475} C_VEL
LIN {X 0,Y 486.875,Z 368.866,A -85,B 0,C 180,E1 21616.096,E2 21616.096} C_VEL
LIN {X 0,Y 483.08,Z 366.683,A -85,B 0,C 180,E1 21613.648,E2 21613.648} C_VEL
LIN {X 0,Y 481.007,Z 363.158,A -85,B 0,C 180,E1 21611.754,E2 21611.754} C_VEL
LIN {X 0,Y 480.724,Z 362.094,A -85,B 0,C 180,E1 21611.397,E2 21611.397} C_VEL
LIN {X 0,Y 476.584,Z 360.089,A -85,B 0,C 180,E1 21604.211,E2 21604.211} C_VEL
LIN {X 0,Y 477.255,Z 360.62,A -85,B 0,C 180,E1 21600.24,E2 21600.24} C_VEL
LIN {X 0,Y 480.776,Z 362.218,A -85,B 0,C 180,E1 21595.646,E2 21595.646} C_VEL
LIN {X 0,Y 482.138,Z 365.496,A -85,B 0,C 180,E1 21594.227,E2 21594.227} C_VEL
LIN {X 0,Y 484.915,Z 368.049,A -85,B 0,C 180,E1 21592.178,E2 21592.178} C_VEL
LIN {X 0,Y 487.086,Z 369.132,A -85,B 0,C 180,E1 21590.876,E2 21590.876} C_VEL
LIN {X 0,Y 488.753,Z 372.474,A -85,B 0,C 180,E1 21589.807,E2 21589.807} C_VEL
LIN {X 0,Y 492.019,Z 375.099,A -85,B 0,C 180,E1 21588.156,E2 21588.156} C_VEL
LIN {X 0,Y 493.062,Z 375.799,A -85,B 0,C 180,E1 21587.676,E2 21587.676} C_VEL
LIN {X 0,Y 495.576,Z 379.759,A -85,B 0,C 180,E1 21586.465,E2 21586.465} C_VEL
LIN {X 0,Y 498.777,Z 382.369,A -85,B 0,C 180,E1 21585.161,E2 21585.161} C_VEL
LIN {X 0,Y 501.425,Z 386.235,A -85,B 0,C 180,E1 21584.086,E2 21584.086} C_VEL
LIN {X 0,Y 504.38,Z 388.868,A -85,B 0,C 180,E1 21583.028,E2 21583.028} C_VEL
LIN {X 0,Y 507.676,Z 393.11,A -85,B 0,C 180,E1 21581.869,E2 21581.869} C_VEL
LIN {X 0,Y 509.655,Z 395.052,A -85,B 0,C 180,E1 21581.231,E2 21581.231} C_VEL
LIN {X 0,Y 513.326,Z 399.578,A -85,B 0,C 180,E1 21580.07,E2 21580.07} C_VEL
LIN {X 0,Y 514.981,Z 401.467,A -85,B 0,C 180,E1 21579.573,E2 21579.573} C_VEL
LIN {X 0,Y 519.026,Z 406.131,A -85,B 0,C 180,E1 21578.41,E2 21578.41} C_VEL
LIN {X 0,Y 525.893,Z 414.789,A -85,B 0,C 180,E1 21576.556,E2 21576.556} C_VEL
LIN {X 0,Y 533.895,Z 425.33,A -85,B 0,C 180,E1 21574.574,E2 21574.574} C_VEL
LIN {X 0,Y 545.508,Z 441.846,A -85,B 0,C 180,E1 21571.956,E2 21571.956} C_VEL
LIN {X 0,Y 558.875,Z 461.903,A -85,B 0,C 180,E1 21569.253,E2 21569.253} C_VEL
LIN {X 0,Y 564.395,Z 470.617,A -85,B 0,C 180,E1 21568.213,E2 21568.213} C_VEL
LIN {X 0,Y 554.631,Z 684.208,A -85,B 0,C 180,E1 21564.995,E2 21564.995} C_VEL
LIN {X 0,Y 548.266,Z 825.818,A -85,B 0,C 180,E1 21562.865,E2 21562.865} C_VEL
LIN {X 0,Y 546.056,Z 852.332,A -85,B 0,C 180,E1 21562.366,E2 21562.366} C_VEL
LIN {X 0,Y 542.811,Z 879.557,A -85,B 0,C 180,E1 21561.662,E2 21561.662} C_VEL
LIN {X 0,Y 539.801,Z 900.633,A -85,B 0,C 180,E1 21560.98,E2 21560.98} C_VEL
LIN {X 0,Y 536.371,Z 921.54,A -85,B 0,C 180,E1 21560.176,E2 21560.176} C_VEL
LIN {X 0,Y 532.593,Z 942.147,A -85,B 0,C 180,E1 21559.245,E2 21559.245} C_VEL
LIN {X 0,Y 527.479,Z 967.328,A -85,B 0,C 180,E1 21557.911,E2 21557.911} C_VEL
LIN {X 0,Y 522.03,Z 991.065,A -85,B 0,C 180,E1 21556.406,E2 21556.406} C_VEL
LIN {X 0,Y 517.567,Z 1009.42,A -85,B 0,C 180,E1 21555.074,E2 21555.074} C_VEL
LIN {X 0,Y 513.028,Z 1027.165,A -85,B 0,C 180,E1 21553.624,E2 21553.624} C_VEL
LIN {X 0,Y 508.265,Z 1045.077,A -85,B 0,C 180,E1 21551.978,E2 21551.978} C_VEL
LIN {X 0,Y 502.317,Z 1066.686,A -85,B 0,C 180,E1 21549.713,E2 21549.713} C_VEL
LIN {X 0,Y 497.247,Z 1084.622,A -85,B 0,C 180,E1 21547.536,E2 21547.536} C_VEL
LIN {X 0,Y 493.204,Z 1098.989,A -85,B 0,C 180,E1 21545.579,E2 21545.579} C_VEL
LIN {X 0,Y 489.371,Z 1112.791,A -85,B 0,C 180,E1 21543.48,E2 21543.48} C_VEL
LIN {X 0,Y 485.58,Z 1126.988,A -85,B 0,C 180,E1 21541.061,E2 21541.061} C_VEL
LIN {X 0,Y 481.412,Z 1143.33,A -85,B 0,C 180,E1 21537.86,E2 21537.86} C_VEL
LIN {X 0,Y 478.708,Z 1154.98,A -85,B 0,C 180,E1 21535.219,E2 21535.219} C_VEL
LIN {X 0,Y 476.665,Z 1164.779,A -85,B 0,C 180,E1 21532.703,E2 21532.703} C_VEL
LIN {X 0,Y 474.937,Z 1174.199,A -85,B 0,C 180,E1 21529.941,E2 21529.941} C_VEL
LIN {X 0,Y 473.411,Z 1184.194,A -85,B 0,C 180,E1 21526.44,E2 21526.44} C_VEL
LIN {X 0,Y 472.691,Z 1190.544,A -85,B 0,C 180,E1 21523.704,E2 21523.704} C_VEL
LIN {X 0,Y 472.249,Z 1195.471,A -85,B 0,C 180,E1 21521.108,E2 21521.108} C_VEL
LIN {X 0,Y 472.048,Z 1199.184,A -85,B 0,C 180,E1 21518.649,E2 21518.649} C_VEL
LIN {X 0,Y 471.949,Z 1201.958,A -85,B 0,C 180,E1 21516.203,E2 21516.203} C_VEL
LIN {X 0,Y 471.915,Z 1203.872,A -85,B 0,C 180,E1 21513.662,E2 21513.662} C_VEL
LIN {X 0,Y 471.913,Z 1204.78,A -85,B 0,C 180,E1 21511.214,E2 21511.214} C_VEL
LIN {X 0,Y 471.913,Z 1204.78,A -85,B 0,C 180,E1 21508.786,E2 21508.786} C_VEL
LIN {X 0,Y 471.915,Z 1203.871,A -85,B 0,C 180,E1 21506.338,E2 21506.338} C_VEL
LIN {X 0,Y 471.949,Z 1201.957,A -85,B 0,C 180,E1 21503.797,E2 21503.797} C_VEL
LIN {X 0,Y 472.056,Z 1199.023,A -85,B 0,C 180,E1 21501.228,E2 21501.228} C_VEL
LIN {X 0,Y 472.296,Z 1194.851,A -85,B 0,C 180,E1 21498.522,E2 21498.522} C_VEL
LIN {X 0,Y 472.952,Z 1188.163,A -85,B 0,C 180,E1 21495.179,E2 21495.179} C_VEL
LIN {X 0,Y 473.92,Z 1180.492,A -85,B 0,C 180,E1 21492.187,E2 21492.187} C_VEL
LIN {X 0,Y 475.207,Z 1172.557,A -85,B 0,C 180,E1 21489.557,E2 21489.557} C_VEL
LIN {X 0,Y 476.885,Z 1163.655,A -85,B 0,C 180,E1 21486.993,E2 21486.993} C_VEL
LIN {X 0,Y 479.307,Z 1152.372,A -85,B 0,C 180,E1 21484.152,E2 21484.152} C_VEL
LIN {X 0,Y 482.784,Z 1137.826,A -85,B 0,C 180,E1 21481.013,E2 21481.013} C_VEL
LIN {X 0,Y 486.175,Z 1124.527,A -85,B 0,C 180,E1 21478.509,E2 21478.509} C_VEL
LIN {X 0,Y 489.79,Z 1111.186,A -85,B 0,C 180,E1 21476.271,E2 21476.271} C_VEL
LIN {X 0,Y 494.524,Z 1094.521,A -85,B 0,C 180,E1 21473.78,E2 21473.78} C_VEL
LIN {X 0,Y 500.092,Z 1075.008,A -85,B 0,C 180,E1 21471.24,E2 21471.24} C_VEL
LIN {X 0,Y 505.018,Z 1057.79,A -85,B 0,C 180,E1 21469.267,E2 21469.267} C_VEL
LIN {X 0,Y 509.747,Z 1041.138,A -85,B 0,C 180,E1 21467.566,E2 21467.566} C_VEL
LIN {X 0,Y 514.704,Z 1023.277,A -85,B 0,C 180,E1 21465.937,E2 21465.937} C_VEL
LIN {X 0,Y 520.816,Z 1000.449,A -85,B 0,C 180,E1 21464.11,E2 21464.11} C_VEL
LIN {X 0,Y 526.501,Z 977.343,A -85,B 0,C 180,E1 21462.538,E2 21462.538} C_VEL
LIN {X 0,Y 530.816,Z 958.764,A -85,B 0,C 180,E1 21461.437,E2 21461.437} C_VEL
LIN {X 0,Y 535.015,Z 938.989,A -85,B 0,C 180,E1 21460.407,E2 21460.407} C_VEL
LIN {X 0,Y 538.985,Z 918.577,A -85,B 0,C 180,E1 21459.492,E2 21459.492} C_VEL
LIN {X 0,Y 543.069,Z 894.932,A -85,B 0,C 180,E1 21458.597,E2 21458.597} C_VEL
LIN {X 0,Y 547.045,Z 866.951,A -85,B 0,C 180,E1 21457.76,E2 21457.76} C_VEL
LIN {X 0,Y 549.586,Z 844.747,A -85,B 0,C 180,E1 21457.245,E2 21457.245} C_VEL
LIN {X 0,Y 551.465,Z 822.53,A -85,B 0,C 180,E1 21456.84,E2 21456.84} C_VEL
LIN {X 0,Y 562.546,Z 606.161,A -85,B 0,C 180,E1 21453.525,E2 21453.525} C_VEL
LIN {X 0,Y 569.786,Z 471.439,A -85,B 0,C 180,E1 21451.445,E2 21451.445} C_VEL
LIN {X 0,Y 562.403,Z 459.784,A -85,B 0,C 180,E1 21449.738,E2 21449.738} C_VEL
LIN {X 0,Y 553.829,Z 446.85,A -85,B 0,C 180,E1 21447.565,E2 21447.565} C_VEL
LIN {X 0,Y 544.79,Z 434.269,A -85,B 0,C 180,E1 21444.999,E2 21444.999} C_VEL
LIN {X 0,Y 538.894,Z 426.267,A -85,B 0,C 180,E1 21443.106,E2 21443.106} C_VEL
LIN {X 0,Y 534.232,Z 420.509,A -85,B 0,C 180,E1 21441.463,E2 21441.463} C_VEL
LIN {X 0,Y 530.548,Z 415.921,A -85,B 0,C 180,E1 21440.031,E2 21440.031} C_VEL
LIN {X 0,Y 526.192,Z 411.037,A -85,B 0,C 180,E1 21438.158,E2 21438.158} C_VEL
LIN {X 0,Y 524.885,Z 409.082,A -85,B 0,C 180,E1 21437.517,E2 21437.517} C_VEL
LIN {X 0,Y 521.314,Z 405.587,A -85,B 0,C 180,E1 21435.691,E2 21435.691} C_VEL
LIN {X 0,Y 519.736,Z 402.988,A -85,B 0,C 180,E1 21434.711,E2 21434.711} C_VEL
LIN {X 0,Y 516.423,Z 400.261,A -85,B 0,C 180,E1 21432.524,E2 21432.524} C_VEL
LIN {X 0,Y 514.624,Z 396.775,A -85,B 0,C 180,E1 21430.863,E2 21430.863} C_VEL
LIN {X 0,Y 510.6,Z 393.996,A -85,B 0,C 180,E1 21424.493,E2 21424.493} C_VEL
LIN {X 0,Y 510.794,Z 394.133,A -85,B 0,C 180,E1 21421.458,E2 21421.458} C_VEL
LIN {X 0,Y 514.623,Z 396.762,A -85,B 0,C 180,E1 21415.933,E2 21415.933} C_VEL
LIN {X 0,Y 516.34,Z 400.181,A -85,B 0,C 180,E1 21414.332,E2 21414.332} C_VEL
LIN {X 0,Y 519.627,Z 402.899,A -85,B 0,C 180,E1 21412.148,E2 21412.148} C_VEL
LIN {X 0,Y 520.324,Z 403.867,A -85,B 0,C 180,E1 21411.713,E2 21411.713} C_VEL
LIN {X 0,Y 522.966,Z 407.56,A -85,B 0,C 180,E1 21410.203,E2 21410.203} C_VEL
LIN {X 0,Y 525.511,Z 409.834,A -85,B 0,C 180,E1 21408.976,E2 21408.976} C_VEL
LIN {X 0,Y 528.622,Z 414.019,A -85,B 0,C 180,E1 21407.547,E2 21407.547} C_VEL
LIN {X 0,Y 530.549,Z 415.919,A -85,B 0,C 180,E1 21406.763,E2 21406.763} C_VEL
LIN {X 0,Y 534.144,Z 420.439,A -85,B 0,C 180,E1 21405.362,E2 21405.362} C_VEL
LIN {X 0,Y 535.768,Z 422.393,A -85,B 0,C 180,E1 21404.771,E2 21404.771} C_VEL
LIN {X 0,Y 540.473,Z 428.176,A -85,B 0,C 180,E1 21403.17,E2 21403.17} C_VEL
LIN {X 0,Y 545.116,Z 434.043,A -85,B 0,C 180,E1 21401.72,E2 21401.72} C_VEL
LIN {X 0,Y 552.032,Z 442.822,A -85,B 0,C 180,E1 21399.76,E2 21399.76} C_VEL
LIN {X 0,Y 561.59,Z 455.892,A -85,B 0,C 180,E1 21397.327,E2 21397.327} C_VEL
LIN {X 0,Y 569.809,Z 468.722,A -85,B 0,C 180,E1 21395.416,E2 21395.416} C_VEL
LIN {X 0,Y 558.389,Z 682.981,A -85,B 0,C 180,E1 21392.123,E2 21392.123} C_VEL
LIN {X 0,Y 551.392,Z 818.824,A -85,B 0,C 180,E1 21390.037,E2 21390.037} C_VEL
LIN {X 0,Y 549.001,Z 845.475,A -85,B 0,C 180,E1 21389.524,E2 21389.524} C_VEL
LIN {X 0,Y 545.548,Z 872.455,A -85,B 0,C 180,E1 21388.81,E2 21388.81} C_VEL
LIN {X 0,Y 542.303,Z 893.719,A -85,B 0,C 180,E1 21388.107,E2 21388.107} C_VEL
LIN {X 0,Y 538.757,Z 913.942,A -85,B 0,C 180,E1 21387.311,E2 21387.311} C_VEL
LIN {X 0,Y 534.591,Z 935.107,A -85,B 0,C 180,E1 21386.335,E2 21386.335} C_VEL
LIN {X 0,Y 528.92,Z 960.996,A -85,B 0,C 180,E1 21384.922,E2 21384.922} C_VEL
LIN {X 0,Y 523.593,Z 982.775,A -85,B 0,C 180,E1 21383.508,E2 21383.508} C_VEL
LIN {X 0,Y 518.743,Z 1001.501,A -85,B 0,C 180,E1 21382.12,E2 21382.12} C_VEL
LIN {X 0,Y 513.92,Z 1019.264,A -85,B 0,C 180,E1 21380.634,E2 21380.634} C_VEL
LIN {X 0,Y 508.779,Z 1037.576,A -85,B 0,C 180,E1 21378.908,E2 21378.908} C_VEL
LIN {X 0,Y 502.175,Z 1060.268,A -85,B 0,C 180,E1 21376.447,E2 21376.447} C_VEL
LIN {X 0,Y 497.356,Z 1076.72,A -85,B 0,C 180,E1 21374.395,E2 21374.395} C_VEL
LIN {X 0,Y 493.043,Z 1091.583,A -85,B 0,C 180,E1 21372.32,E2 21372.32} C_VEL
LIN {X 0,Y 488.381,Z 1108.303,A -85,B 0,C 180,E1 21369.699,E2 21369.699} C_VEL
LIN {X 0,Y 487.599,Z 1111.019,A -85,B 0,C 180,E1 21369.234,E2 21369.234} C_VEL
LIN {X 0,Y 485.465,Z 1115.443,A -85,B 0,C 180,E1 21368.519,E2 21368.519} C_VEL
LIN {X 0,Y 476.693,Z 1127.212,A -85,B 0,C 180,E1 21366.69,E2 21366.69} C_VEL
LIN {X 0,Y 475.09,Z 1130.636,A -85,B 0,C 180,E1 21366.035,E2 21366.035} C_VEL
LIN {X 0,Y 471.512,Z 1144.524,A -85,B 0,C 180,E1 21362.878,E2 21362.878} C_VEL
LIN {X 0,Y 468.956,Z 1155.721,A -85,B 0,C 180,E1 21359.928,E2 21359.928} C_VEL
LIN {X 0,Y 466.962,Z 1165.691,A -85,B 0,C 180,E1 21356.859,E2 21356.859} C_VEL
LIN {X 0,Y 465.452,Z 1175.027,A -85,B 0,C 180,E1 21353.416,E2 21353.416} C_VEL
LIN {X 0,Y 464.644,Z 1181.613,A -85,B 0,C 180,E1 21350.402,E2 21350.402} C_VEL
LIN {X 0,Y 464.232,Z 1186.22,A -85,B 0,C 180,E1 21347.809,E2 21347.809} C_VEL
LIN {X 0,Y 464.028,Z 1189.992,A -85,B 0,C 180,E1 21345.113,E2 21345.113} C_VEL
LIN {X 0,Y 463.933,Z 1192.919,A -85,B 0,C 180,E1 21342.193,E2 21342.193} C_VEL
LIN {X 0,Y 463.911,Z 1194.654,A -85,B 0,C 180,E1 21338.927,E2 21338.927} C_VEL
LIN {X 0,Y 463.914,Z 1194.847,A -85,B 0,C 180,E1 21336.062,E2 21336.062} C_VEL
LIN {X 0,Y 463.913,Z 1193.999,A -85,B 0,C 180,E1 21333.46,E2 21333.46} C_VEL
LIN {X 0,Y 463.948,Z 1192.161,A -85,B 0,C 180,E1 21330.864,E2 21330.864} C_VEL
LIN {X 0,Y 464.051,Z 1189.339,A -85,B 0,C 180,E1 21328.271,E2 21328.271} C_VEL
LIN {X 0,Y 464.335,Z 1184.961,A -85,B 0,C 180,E1 21325.307,E2 21325.307} C_VEL
LIN {X 0,Y 465.038,Z 1178.134,A -85,B 0,C 180,E1 21321.842,E2 21321.842} C_VEL
LIN {X 0,Y 466.028,Z 1171.147,A -85,B 0,C 180,E1 21318.992,E2 21318.992} C_VEL
LIN {X 0,Y 467.491,Z 1162.892,A -85,B 0,C 180,E1 21316.141,E2 21316.141} C_VEL
LIN {X 0,Y 469.994,Z 1150.974,A -85,B 0,C 180,E1 21312.673,E2 21312.673} C_VEL
LIN {X 0,Y 473.171,Z 1137.836,A -85,B 0,C 180,E1 21309.465,E2 21309.465} C_VEL
LIN {X 0,Y 476.511,Z 1125.111,A -85,B 0,C 180,E1 21306.767,E2 21306.767} C_VEL
LIN {X 0,Y 481.022,Z 1109.44,A -85,B 0,C 180,E1 21303.854,E2 21303.854} C_VEL
LIN {X 0,Y 485.816,Z 1092.837,A -85,B 0,C 180,E1 21301.21,E2 21301.21} C_VEL
LIN {X 0,Y 490.312,Z 1077.667,A -85,B 0,C 180,E1 21299.077,E2 21299.077} C_VEL
LIN {X 0,Y 494.867,Z 1062.271,A -85,B 0,C 180,E1 21297.147,E2 21297.147} C_VEL
LIN {X 0,Y 500.331,Z 1043.62,A -85,B 0,C 180,E1 21295.073,E2 21295.073} C_VEL
LIN {X 0,Y 506.468,Z 1021.788,A -85,B 0,C 180,E1 21292.978,E2 21292.978} C_VEL
LIN {X 0,Y 511.446,Z 1003.167,A -85,B 0,C 180,E1 21291.418,E2 21291.418} C_VEL
LIN {X 0,Y 516.076,Z 984.931,A -85,B 0,C 180,E1 21290.067,E2 21290.067} C_VEL
LIN {X 0,Y 520.693,Z 965.592,A -85,B 0,C 180,E1 21288.804,E2 21288.804} C_VEL
LIN {X 0,Y 525.88,Z 942.143,A -85,B 0,C 180,E1 21287.475,E2 21287.475} C_VEL
LIN {X 0,Y 530.811,Z 916.514,A -85,B 0,C 180,E1 21286.267,E2 21286.267} C_VEL
LIN {X 0,Y 534.374,Z 895.604,A -85,B 0,C 180,E1 21285.44,E2 21285.44} C_VEL
LIN {X 0,Y 537.452,Z 874.751,A -85,B 0,C 180,E1 21284.745,E2 21284.745} C_VEL
LIN {X 0,Y 540.234,Z 852.58,A -85,B 0,C 180,E1 21284.14,E2 21284.14} C_VEL
LIN {X 0,Y 542.928,Z 825.364,A -85,B 0,C 180,E1 21283.566,E2 21283.566} C_VEL
LIN {X 0,Y 545.275,Z 780.262,A -85,B 0,C 180,E1 21282.863,E2 21282.863} C_VEL
LIN {X 0,Y 555.635,Z 556.383,A -85,B 0,C 180,E1 21279.494,E2 21279.494} C_VEL
LIN {X 0,Y 559.594,Z 471.71,A -85,B 0,C 180,E1 21278.188,E2 21278.188} C_VEL
LIN {X 0,Y 548.326,Z 454.656,A -85,B 0,C 180,E1 21275.957,E2 21275.957} C_VEL
LIN {X 0,Y 536.645,Z 438.827,A -85,B 0,C 180,E1 21273.439,E2 21273.439} C_VEL
LIN {X 0,Y 528.1,Z 427.788,A -85,B 0,C 180,E1 21271.41,E2 21271.41} C_VEL
LIN {X 0,Y 520.686,Z 418.291,A -85,B 0,C 180,E1 21269.478,E2 21269.478} C_VEL
LIN {X 0,Y 515.967,Z 412.572,A -85,B 0,C 180,E1 21268.156,E2 21268.156} C_VEL
LIN {X 0,Y 511.58,Z 407.175,A -85,B 0,C 180,E1 21266.84,E2 21266.84} C_VEL
LIN {X 0,Y 507.667,Z 402.372,A -85,B 0,C 180,E1 21265.584,E2 21265.584} C_VEL
LIN {X 0,Y 503.229,Z 397.466,A -85,B 0,C 180,E1 21264.068,E2 21264.068} C_VEL
LIN {X 0,Y 501.825,Z 395.621,A -85,B 0,C 180,E1 21263.547,E2 21263.547} C_VEL
LIN {X 0,Y 498.334,Z 392.003,A -85,B 0,C 180,E1 21262.224,E2 21262.224} C_VEL
LIN {X 0,Y 496.903,Z 389.624,A -85,B 0,C 180,E1 21261.607,E2 21261.607} C_VEL
LIN {X 0,Y 493.444,Z 386.657,A -85,B 0,C 180,E1 21260.15,E2 21260.15} C_VEL
LIN {X 0,Y 491.138,Z 383.164,A -85,B 0,C 180,E1 21259.01,E2 21259.01} C_VEL
LIN {X 0,Y 487.819,Z 380.749,A -85,B 0,C 180,E1 21257.352,E2 21257.352} C_VEL
LIN {X 0,Y 485.831,Z 377.231,A -85,B 0,C 180,E1 21256.101,E2 21256.101} C_VEL
LIN {X 0,Y 485.321,Z 376.649,A -85,B 0,C 180,E1 21255.781,E2 21255.781} C_VEL
LIN {X 0,Y 481.813,Z 374.413,A -85,B 0,C 180,E1 21253.44,E2 21253.44} C_VEL
LIN {X 0,Y 479.798,Z 370.877,A -85,B 0,C 180,E1 21251.541,E2 21251.541} C_VEL
LIN {X 0,Y 479.504,Z 369.982,A -85,B 0,C 180,E1 21251.182,E2 21251.182} C_VEL
LIN {X 0,Y 475.609,Z 368.029,A -85,B 0,C 180,E1 21244.22,E2 21244.22} C_VEL
LIN {X 0,Y 476.276,Z 368.566,A -85,B 0,C 180,E1 21240.241,E2 21240.241} C_VEL
LIN {X 0,Y 479.602,Z 370.128,A -85,B 0,C 180,E1 21235.815,E2 21235.815} C_VEL
LIN {X 0,Y 481.213,Z 373.69,A -85,B 0,C 180,E1 21234.156,E2 21234.156} C_VEL
LIN {X 0,Y 484.497,Z 376.32,A -85,B 0,C 180,E1 21231.813,E2 21231.813} C_VEL
LIN {X 0,Y 485.748,Z 377.062,A -85,B 0,C 180,E1 21231.059,E2 21231.059} C_VEL
LIN {X 0,Y 487.66,Z 380.525,A -85,B 0,C 180,E1 21229.844,E2 21229.844} C_VEL
LIN {X 0,Y 491.056,Z 383.089,A -85,B 0,C 180,E1 21228.132,E2 21228.132} C_VEL
LIN {X 0,Y 491.746,Z 383.943,A -85,B 0,C 180,E1 21227.792,E2 21227.792} C_VEL
LIN {X 0,Y 494.594,Z 387.961,A -85,B 0,C 180,E1 21226.437,E2 21226.437} C_VEL
LIN {X 0,Y 497.163,Z 390.097,A -85,B 0,C 180,E1 21225.38,E2 21225.38} C_VEL
LIN {X 0,Y 500.154,Z 394.206,A -85,B 0,C 180,E1 21224.164,E2 21224.164} C_VEL
LIN {X 0,Y 502.63,Z 396.473,A -85,B 0,C 180,E1 21223.264,E2 21223.264} C_VEL
LIN {X 0,Y 506.055,Z 400.789,A -85,B 0,C 180,E1 21222.047,E2 21222.047} C_VEL
LIN {X 0,Y 507.839,Z 402.67,A -85,B 0,C 180,E1 21221.459,E2 21221.459} C_VEL
LIN {X 0,Y 511.658,Z 407.263,A -85,B 0,C 180,E1 21220.24,E2 21220.24} C_VEL
LIN {X 0,Y 518.1,Z 415.128,A -85,B 0,C 180,E1 21218.34,E2 21218.34} C_VEL
LIN {X 0,Y 523.063,Z 421.291,A -85,B 0,C 180,E1 21216.988,E2 21216.988} C_VEL
LIN {X 0,Y 530.027,Z 430.56,A -85,B 0,C 180,E1 21215.211,E2 21215.211} C_VEL
LIN {X 0,Y 541.315,Z 446.589,A -85,B 0,C 180,E1 21212.587,E2 21212.587} C_VEL
LIN {X 0,Y 555.025,Z 467.313,A -85,B 0,C 180,E1 21209.736,E2 21209.736} C_VEL
LIN {X 0,Y 559.698,Z 474.956,A -85,B 0,C 180,E1 21208.827,E2 21208.827} C_VEL
